// SIMATIC STEP 7 (V5.x) project cc1_15_7_14
// CPU: CPU 315-2 DP
// station: P_ADR_BUS
// station: Hardware
// station: SIMATIC 300 - BEC
// program: S7 Program(1)

FUNCTION FC 1 : VOID
AUTHOR : Arun
VERSION : 0.1
BEGIN
// (block stored without names or comments; labels and parameter names are numbered)
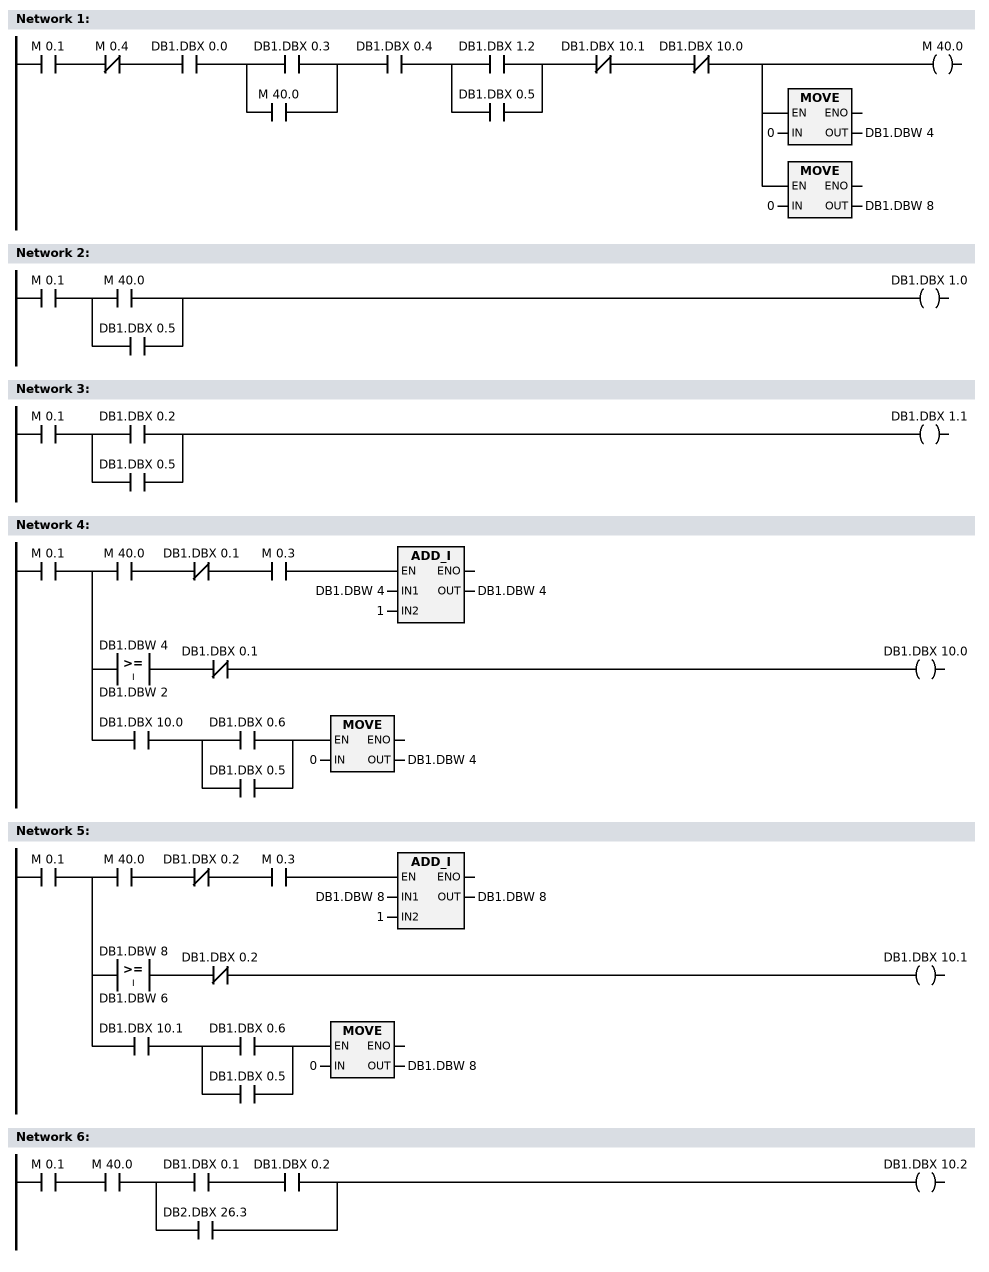
NETWORK
TITLE =
      A     M 0.1;
      AN    M 0.4;
      A     DB1.DBX 0.0;
      A(;
      O     DB1.DBX 0.3;
      O     M 40.0;
      );
      A     DB1.DBX 0.4;
      A(;
      O     DB1.DBX 1.2;
      O     DB1.DBX 0.5;
      );
      AN    DB1.DBX 10.1;
      AN    DB1.DBX 10.0;
      =     L 0.0;
      A     L 0.0;
      BLD   102;
      =     M 40.0;
      A     L 0.0;
      JNB   M001;
      L     0;
      T     DB1.DBW 4;
M001: NOP   0;
      A     L 0.0;
      JNB   M002;
      L     0;
      T     DB1.DBW 8;
M002: NOP   0;
NETWORK
TITLE =
      A     M 0.1;
      A(;
      O     M 40.0;
      O     DB1.DBX 0.5;
      );
      =     DB1.DBX 1.0;
NETWORK
TITLE =
      A     M 0.1;
      A(;
      O     DB1.DBX 0.2;
      O     DB1.DBX 0.5;
      );
      =     DB1.DBX 1.1;
NETWORK
TITLE =
      A     M 0.1;
      =     L 0.0;
      A     L 0.0;
      A     M 40.0;
      AN    DB1.DBX 0.1;
      A     M 0.3;
      JNB   M003;
      L     DB1.DBW 4;
      L     1;
      +I;
      T     DB1.DBW 4;
M003: NOP   0;
      A     L 0.0;
      A(;
      L     DB1.DBW 4;
      L     DB1.DBW 2;
      >=I;
      );
      AN    DB1.DBX 0.1;
      =     DB1.DBX 10.0;
      A     L 0.0;
      A     DB1.DBX 10.0;
      A(;
      O     DB1.DBX 0.6;
      O     DB1.DBX 0.5;
      );
      JNB   M004;
      L     0;
      T     DB1.DBW 4;
M004: NOP   0;
NETWORK
TITLE =
      A     M 0.1;
      =     L 0.0;
      A     L 0.0;
      A     M 40.0;
      AN    DB1.DBX 0.2;
      A     M 0.3;
      JNB   M005;
      L     DB1.DBW 8;
      L     1;
      +I;
      T     DB1.DBW 8;
M005: NOP   0;
      A     L 0.0;
      A(;
      L     DB1.DBW 8;
      L     DB1.DBW 6;
      >=I;
      );
      AN    DB1.DBX 0.2;
      =     DB1.DBX 10.1;
      A     L 0.0;
      A     DB1.DBX 10.1;
      A(;
      O     DB1.DBX 0.6;
      O     DB1.DBX 0.5;
      );
      JNB   M006;
      L     0;
      T     DB1.DBW 8;
M006: NOP   0;
NETWORK
TITLE =
      A     M 0.1;
      A     M 40.0;
      A(;
      A     DB1.DBX 0.1;
      A     DB1.DBX 0.2;
      O     DB2.DBX 26.3;
      );
      =     DB1.DBX 10.2;
END_FUNCTION

// FC 2: know-how protected block, not included

// FC 3: know-how protected block, not included

// FC 4: know-how protected block, not included

FUNCTION FC 5 : VOID
AUTHOR : Arun_Ram
VERSION : 0.1
BEGIN
// (block stored without names or comments; labels and parameter names are numbered)
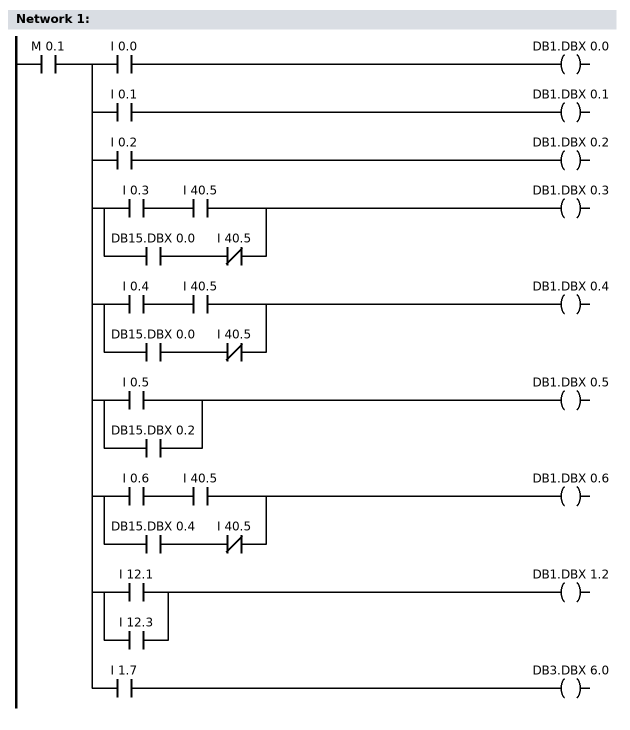
NETWORK
TITLE =
      A     M 0.1;
      =     L 0.0;
      A     L 0.0;
      A     I 0.0;
      =     DB1.DBX 0.0;
      A     L 0.0;
      A     I 0.1;
      =     DB1.DBX 0.1;
      A     L 0.0;
      A     I 0.2;
      =     DB1.DBX 0.2;
      A     L 0.0;
      A(;
      A     I 0.3;
      A     I 40.5;
      O;
      A     DB15.DBX 0.0;
      AN    I 40.5;
      );
      =     DB1.DBX 0.3;
      A     L 0.0;
      A(;
      A     I 0.4;
      A     I 40.5;
      O;
      A     DB15.DBX 0.0;
      AN    I 40.5;
      );
      =     DB1.DBX 0.4;
      A     L 0.0;
      A(;
      O     I 0.5;
      O     DB15.DBX 0.2;
      );
      =     DB1.DBX 0.5;
      A     L 0.0;
      A(;
      A     I 0.6;
      A     I 40.5;
      O;
      A     DB15.DBX 0.4;
      AN    I 40.5;
      );
      =     DB1.DBX 0.6;
      A     L 0.0;
      A(;
      O     I 12.1;
      O     I 12.3;
      );
      =     DB1.DBX 1.2;
      A     L 0.0;
      A     I 1.7;
      =     DB3.DBX 6.0;
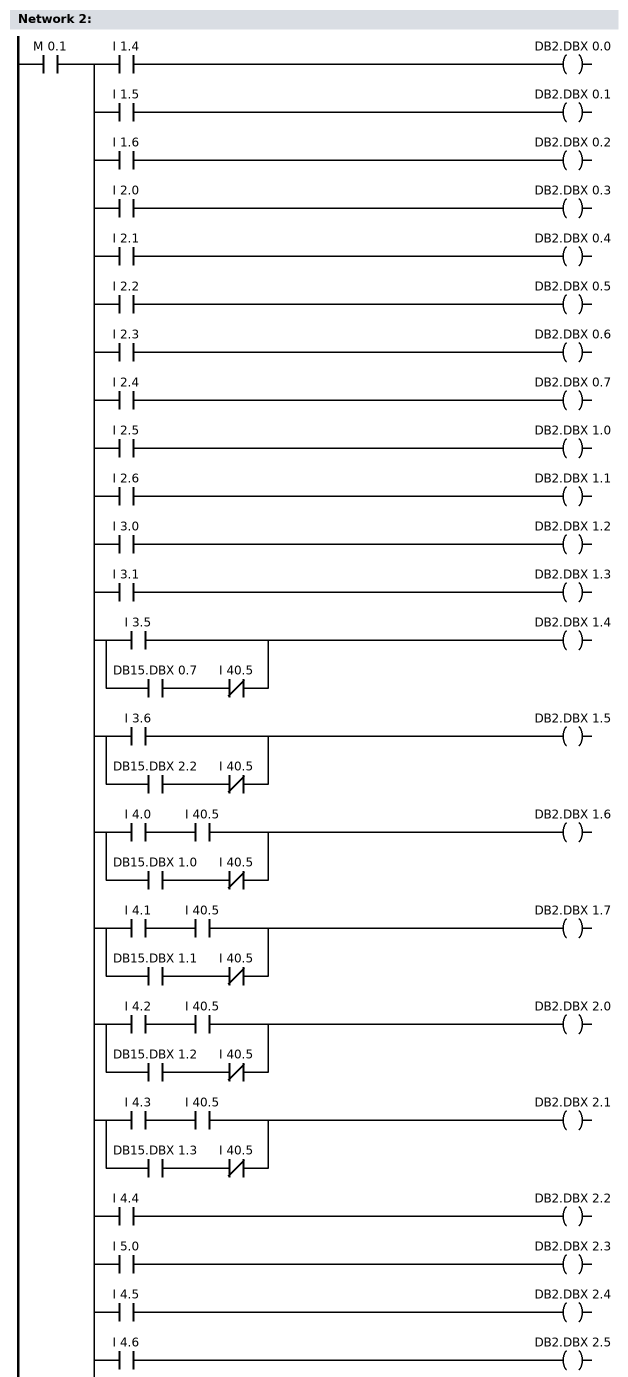
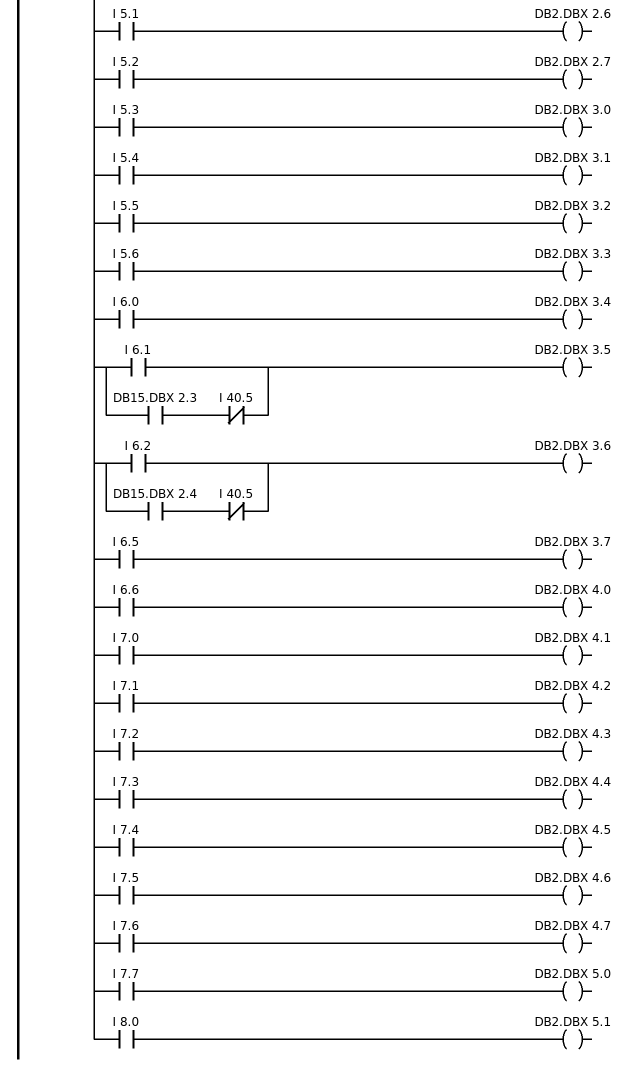
NETWORK
TITLE =
      A     M 0.1;
      =     L 0.0;
      A     L 0.0;
      A     I 1.4;
      =     DB2.DBX 0.0;
      A     L 0.0;
      A     I 1.5;
      =     DB2.DBX 0.1;
      A     L 0.0;
      A     I 1.6;
      =     DB2.DBX 0.2;
      A     L 0.0;
      A     I 2.0;
      =     DB2.DBX 0.3;
      A     L 0.0;
      A     I 2.1;
      =     DB2.DBX 0.4;
      A     L 0.0;
      A     I 2.2;
      =     DB2.DBX 0.5;
      A     L 0.0;
      A     I 2.3;
      =     DB2.DBX 0.6;
      A     L 0.0;
      A     I 2.4;
      =     DB2.DBX 0.7;
      A     L 0.0;
      A     I 2.5;
      =     DB2.DBX 1.0;
      A     L 0.0;
      A     I 2.6;
      =     DB2.DBX 1.1;
      A     L 0.0;
      A     I 3.0;
      =     DB2.DBX 1.2;
      A     L 0.0;
      A     I 3.1;
      =     DB2.DBX 1.3;
      A     L 0.0;
      A(;
      O     I 3.5;
      O;
      A     DB15.DBX 0.7;
      AN    I 40.5;
      );
      =     DB2.DBX 1.4;
      A     L 0.0;
      A(;
      O     I 3.6;
      O;
      A     DB15.DBX 2.2;
      AN    I 40.5;
      );
      =     DB2.DBX 1.5;
      A     L 0.0;
      A(;
      A     I 4.0;
      A     I 40.5;
      O;
      A     DB15.DBX 1.0;
      AN    I 40.5;
      );
      =     DB2.DBX 1.6;
      A     L 0.0;
      A(;
      A     I 4.1;
      A     I 40.5;
      O;
      A     DB15.DBX 1.1;
      AN    I 40.5;
      );
      =     DB2.DBX 1.7;
      A     L 0.0;
      A(;
      A     I 4.2;
      A     I 40.5;
      O;
      A     DB15.DBX 1.2;
      AN    I 40.5;
      );
      =     DB2.DBX 2.0;
      A     L 0.0;
      A(;
      A     I 4.3;
      A     I 40.5;
      O;
      A     DB15.DBX 1.3;
      AN    I 40.5;
      );
      =     DB2.DBX 2.1;
      A     L 0.0;
      A     I 4.4;
      =     DB2.DBX 2.2;
      A     L 0.0;
      A     I 5.0;
      =     DB2.DBX 2.3;
      A     L 0.0;
      A     I 4.5;
      =     DB2.DBX 2.4;
      A     L 0.0;
      A     I 4.6;
      =     DB2.DBX 2.5;
      A     L 0.0;
      A     I 5.1;
      =     DB2.DBX 2.6;
      A     L 0.0;
      A     I 5.2;
      =     DB2.DBX 2.7;
      A     L 0.0;
      A     I 5.3;
      =     DB2.DBX 3.0;
      A     L 0.0;
      A     I 5.4;
      =     DB2.DBX 3.1;
      A     L 0.0;
      A     I 5.5;
      =     DB2.DBX 3.2;
      A     L 0.0;
      A     I 5.6;
      =     DB2.DBX 3.3;
      A     L 0.0;
      A     I 6.0;
      =     DB2.DBX 3.4;
      A     L 0.0;
      A(;
      O     I 6.1;
      O;
      A     DB15.DBX 2.3;
      AN    I 40.5;
      );
      =     DB2.DBX 3.5;
      A     L 0.0;
      A(;
      O     I 6.2;
      O;
      A     DB15.DBX 2.4;
      AN    I 40.5;
      );
      =     DB2.DBX 3.6;
      A     L 0.0;
      A     I 6.5;
      =     DB2.DBX 3.7;
      A     L 0.0;
      A     I 6.6;
      =     DB2.DBX 4.0;
      A     L 0.0;
      A     I 7.0;
      =     DB2.DBX 4.1;
      A     L 0.0;
      A     I 7.1;
      =     DB2.DBX 4.2;
      A     L 0.0;
      A     I 7.2;
      =     DB2.DBX 4.3;
      A     L 0.0;
      A     I 7.3;
      =     DB2.DBX 4.4;
      A     L 0.0;
      A     I 7.4;
      =     DB2.DBX 4.5;
      A     L 0.0;
      A     I 7.5;
      =     DB2.DBX 4.6;
      A     L 0.0;
      A     I 7.6;
      =     DB2.DBX 4.7;
      A     L 0.0;
      A     I 7.7;
      =     DB2.DBX 5.0;
      A     L 0.0;
      A     I 8.0;
      =     DB2.DBX 5.1;
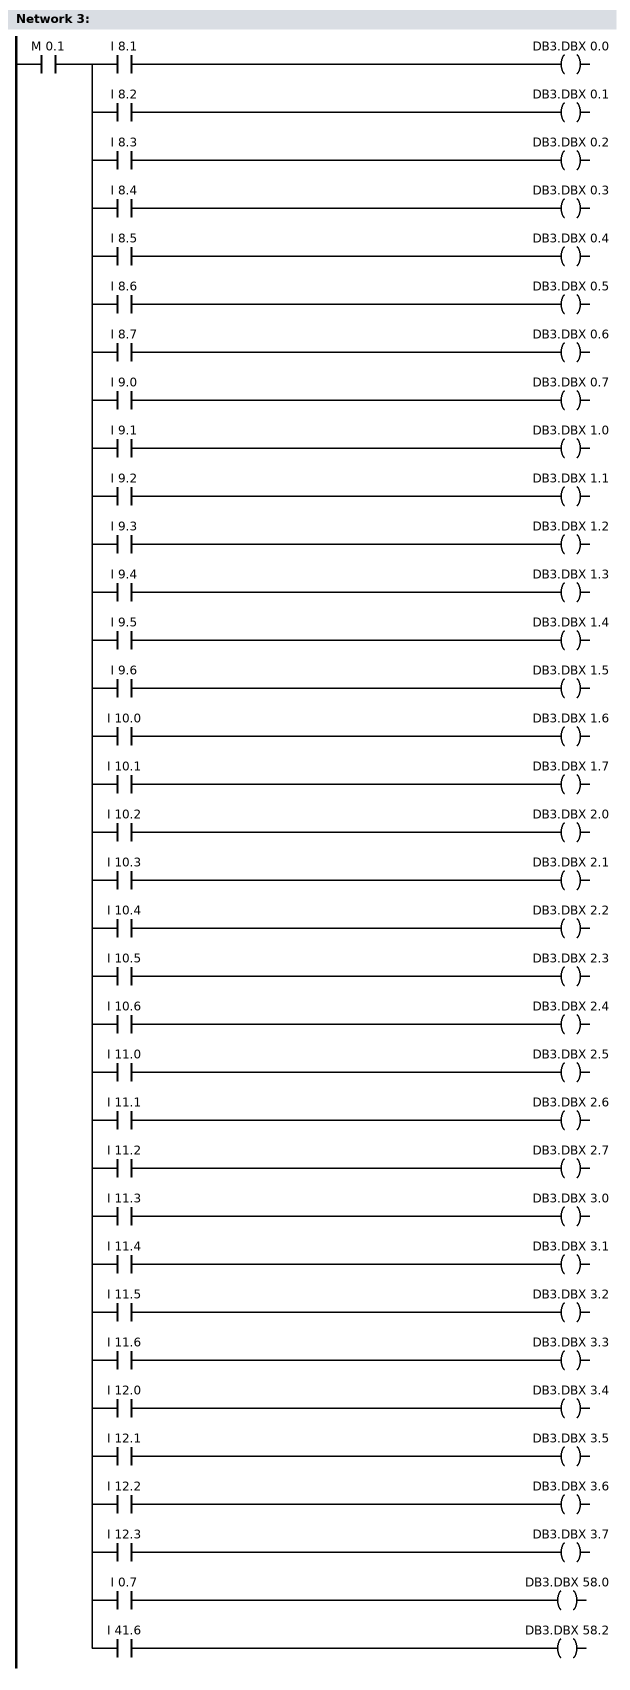
NETWORK
TITLE =
      A     M 0.1;
      =     L 0.0;
      A     L 0.0;
      A     I 8.1;
      =     DB3.DBX 0.0;
      A     L 0.0;
      A     I 8.2;
      =     DB3.DBX 0.1;
      A     L 0.0;
      A     I 8.3;
      =     DB3.DBX 0.2;
      A     L 0.0;
      A     I 8.4;
      =     DB3.DBX 0.3;
      A     L 0.0;
      A     I 8.5;
      =     DB3.DBX 0.4;
      A     L 0.0;
      A     I 8.6;
      =     DB3.DBX 0.5;
      A     L 0.0;
      A     I 8.7;
      =     DB3.DBX 0.6;
      A     L 0.0;
      A     I 9.0;
      =     DB3.DBX 0.7;
      A     L 0.0;
      A     I 9.1;
      =     DB3.DBX 1.0;
      A     L 0.0;
      A     I 9.2;
      =     DB3.DBX 1.1;
      A     L 0.0;
      A     I 9.3;
      =     DB3.DBX 1.2;
      A     L 0.0;
      A     I 9.4;
      =     DB3.DBX 1.3;
      A     L 0.0;
      A     I 9.5;
      =     DB3.DBX 1.4;
      A     L 0.0;
      A     I 9.6;
      =     DB3.DBX 1.5;
      A     L 0.0;
      A     I 10.0;
      =     DB3.DBX 1.6;
      A     L 0.0;
      A     I 10.1;
      =     DB3.DBX 1.7;
      A     L 0.0;
      A     I 10.2;
      =     DB3.DBX 2.0;
      A     L 0.0;
      A     I 10.3;
      =     DB3.DBX 2.1;
      A     L 0.0;
      A     I 10.4;
      =     DB3.DBX 2.2;
      A     L 0.0;
      A     I 10.5;
      =     DB3.DBX 2.3;
      A     L 0.0;
      A     I 10.6;
      =     DB3.DBX 2.4;
      A     L 0.0;
      A     I 11.0;
      =     DB3.DBX 2.5;
      A     L 0.0;
      A     I 11.1;
      =     DB3.DBX 2.6;
      A     L 0.0;
      A     I 11.2;
      =     DB3.DBX 2.7;
      A     L 0.0;
      A     I 11.3;
      =     DB3.DBX 3.0;
      A     L 0.0;
      A     I 11.4;
      =     DB3.DBX 3.1;
      A     L 0.0;
      A     I 11.5;
      =     DB3.DBX 3.2;
      A     L 0.0;
      A     I 11.6;
      =     DB3.DBX 3.3;
      A     L 0.0;
      A     I 12.0;
      =     DB3.DBX 3.4;
      A     L 0.0;
      A     I 12.1;
      =     DB3.DBX 3.5;
      A     L 0.0;
      A     I 12.2;
      =     DB3.DBX 3.6;
      A     L 0.0;
      A     I 12.3;
      =     DB3.DBX 3.7;
      A     L 0.0;
      A     I 0.7;
      =     DB3.DBX 58.0;
      A     L 0.0;
      A     I 41.6;
      =     DB3.DBX 58.2;
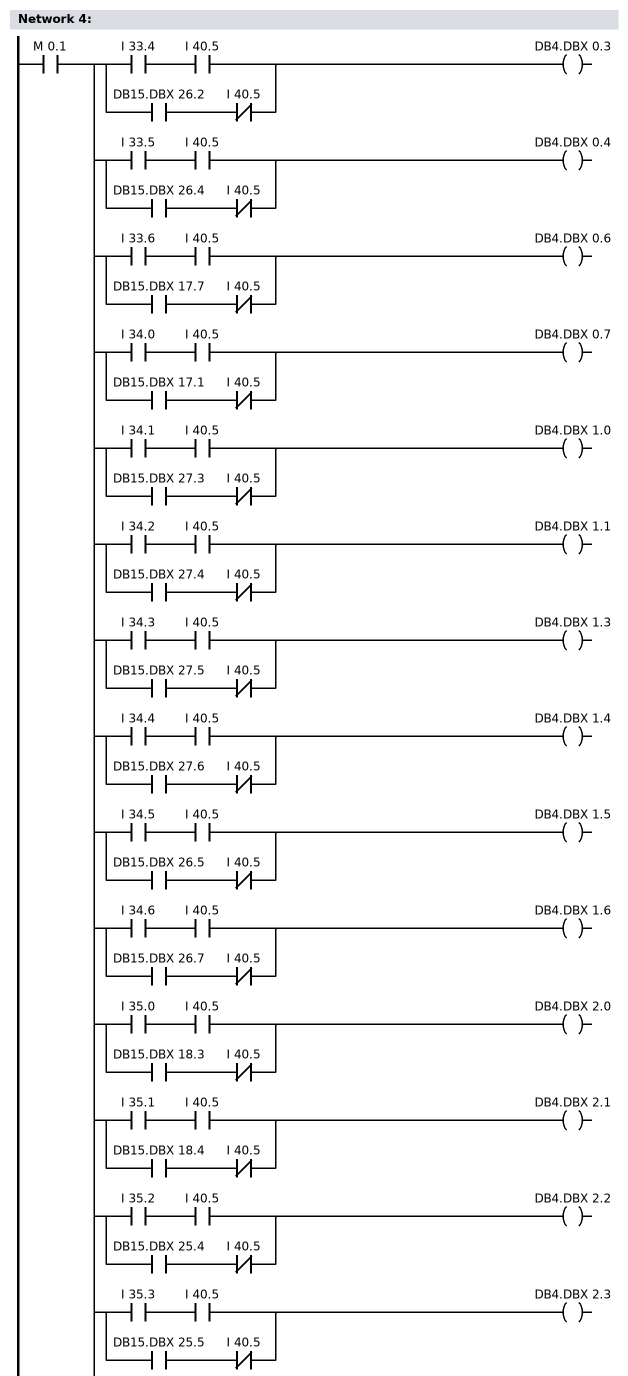
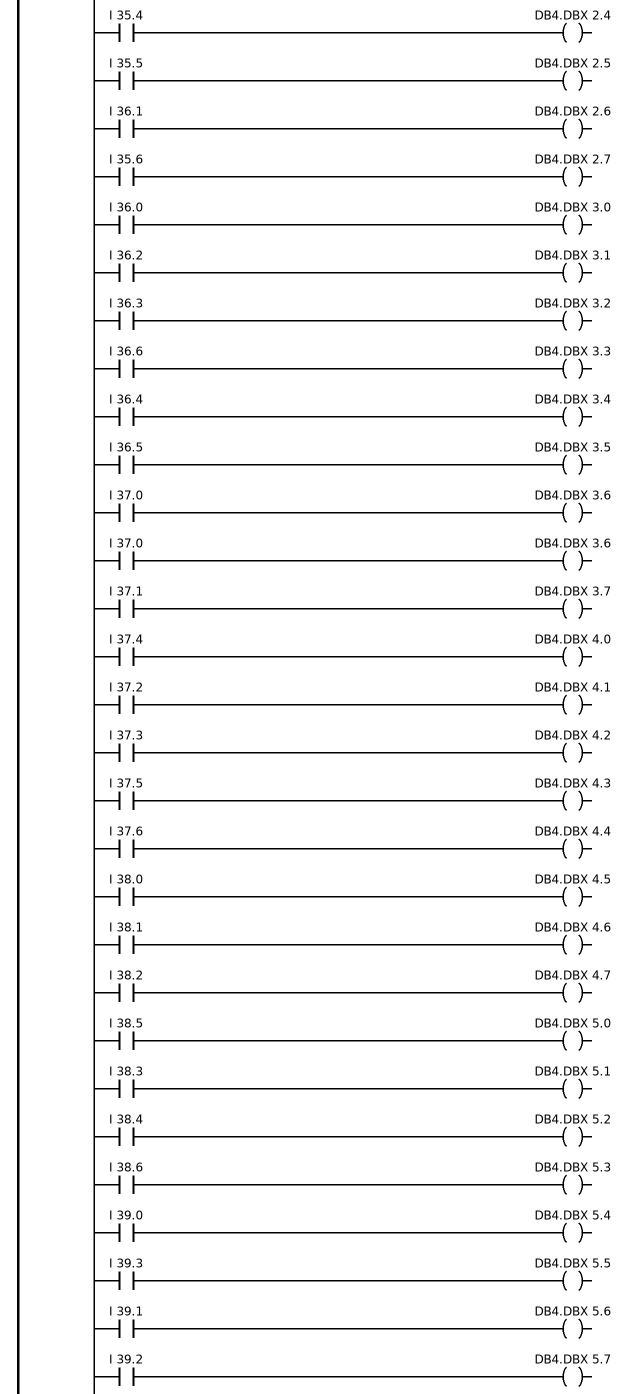
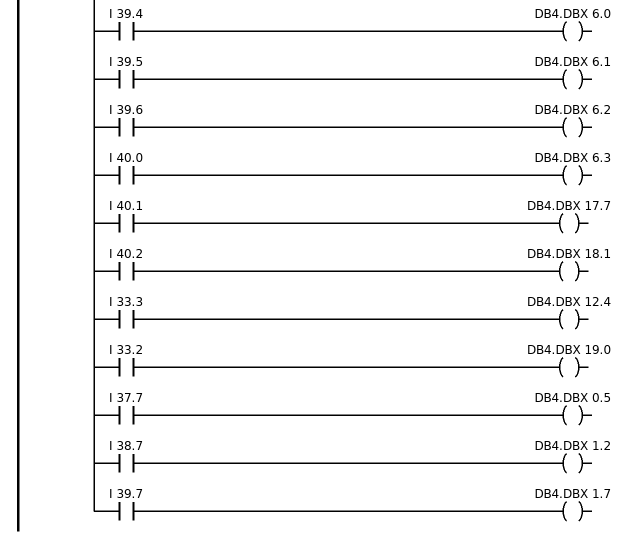
NETWORK
TITLE =
      A     M 0.1;
      =     L 0.0;
      A     L 0.0;
      A(;
      A     I 33.4;
      A     I 40.5;
      O;
      A     DB15.DBX 26.2;
      AN    I 40.5;
      );
      =     DB4.DBX 0.3;
      A     L 0.0;
      A(;
      A     I 33.5;
      A     I 40.5;
      O;
      A     DB15.DBX 26.4;
      AN    I 40.5;
      );
      =     DB4.DBX 0.4;
      A     L 0.0;
      A(;
      A     I 33.6;
      A     I 40.5;
      O;
      A     DB15.DBX 17.7;
      AN    I 40.5;
      );
      =     DB4.DBX 0.6;
      A     L 0.0;
      A(;
      A     I 34.0;
      A     I 40.5;
      O;
      A     DB15.DBX 17.1;
      AN    I 40.5;
      );
      =     DB4.DBX 0.7;
      A     L 0.0;
      A(;
      A     I 34.1;
      A     I 40.5;
      O;
      A     DB15.DBX 27.3;
      AN    I 40.5;
      );
      =     DB4.DBX 1.0;
      A     L 0.0;
      A(;
      A     I 34.2;
      A     I 40.5;
      O;
      A     DB15.DBX 27.4;
      AN    I 40.5;
      );
      =     DB4.DBX 1.1;
      A     L 0.0;
      A(;
      A     I 34.3;
      A     I 40.5;
      O;
      A     DB15.DBX 27.5;
      AN    I 40.5;
      );
      =     DB4.DBX 1.3;
      A     L 0.0;
      A(;
      A     I 34.4;
      A     I 40.5;
      O;
      A     DB15.DBX 27.6;
      AN    I 40.5;
      );
      =     DB4.DBX 1.4;
      A     L 0.0;
      A(;
      A     I 34.5;
      A     I 40.5;
      O;
      A     DB15.DBX 26.5;
      AN    I 40.5;
      );
      =     DB4.DBX 1.5;
      A     L 0.0;
      A(;
      A     I 34.6;
      A     I 40.5;
      O;
      A     DB15.DBX 26.7;
      AN    I 40.5;
      );
      =     DB4.DBX 1.6;
      A     L 0.0;
      A(;
      A     I 35.0;
      A     I 40.5;
      O;
      A     DB15.DBX 18.3;
      AN    I 40.5;
      );
      =     DB4.DBX 2.0;
      A     L 0.0;
      A(;
      A     I 35.1;
      A     I 40.5;
      O;
      A     DB15.DBX 18.4;
      AN    I 40.5;
      );
      =     DB4.DBX 2.1;
      A     L 0.0;
      A(;
      A     I 35.2;
      A     I 40.5;
      O;
      A     DB15.DBX 25.4;
      AN    I 40.5;
      );
      =     DB4.DBX 2.2;
      A     L 0.0;
      A(;
      A     I 35.3;
      A     I 40.5;
      O;
      A     DB15.DBX 25.5;
      AN    I 40.5;
      );
      =     DB4.DBX 2.3;
      A     L 0.0;
      A     I 35.4;
      =     DB4.DBX 2.4;
      A     L 0.0;
      A     I 35.5;
      =     DB4.DBX 2.5;
      A     L 0.0;
      A     I 36.1;
      =     DB4.DBX 2.6;
      A     L 0.0;
      A     I 35.6;
      =     DB4.DBX 2.7;
      A     L 0.0;
      A     I 36.0;
      =     DB4.DBX 3.0;
      A     L 0.0;
      A     I 36.2;
      =     DB4.DBX 3.1;
      A     L 0.0;
      A     I 36.3;
      =     DB4.DBX 3.2;
      A     L 0.0;
      A     I 36.6;
      =     DB4.DBX 3.3;
      A     L 0.0;
      A     I 36.4;
      =     DB4.DBX 3.4;
      A     L 0.0;
      A     I 36.5;
      =     DB4.DBX 3.5;
      A     L 0.0;
      A     I 37.0;
      =     DB4.DBX 3.6;
      A     L 0.0;
      A     I 37.0;
      =     DB4.DBX 3.6;
      A     L 0.0;
      A     I 37.1;
      =     DB4.DBX 3.7;
      A     L 0.0;
      A     I 37.4;
      =     DB4.DBX 4.0;
      A     L 0.0;
      A     I 37.2;
      =     DB4.DBX 4.1;
      A     L 0.0;
      A     I 37.3;
      =     DB4.DBX 4.2;
      A     L 0.0;
      A     I 37.5;
      =     DB4.DBX 4.3;
      A     L 0.0;
      A     I 37.6;
      =     DB4.DBX 4.4;
      A     L 0.0;
      A     I 38.0;
      =     DB4.DBX 4.5;
      A     L 0.0;
      A     I 38.1;
      =     DB4.DBX 4.6;
      A     L 0.0;
      A     I 38.2;
      =     DB4.DBX 4.7;
      A     L 0.0;
      A     I 38.5;
      =     DB4.DBX 5.0;
      A     L 0.0;
      A     I 38.3;
      =     DB4.DBX 5.1;
      A     L 0.0;
      A     I 38.4;
      =     DB4.DBX 5.2;
      A     L 0.0;
      A     I 38.6;
      =     DB4.DBX 5.3;
      A     L 0.0;
      A     I 39.0;
      =     DB4.DBX 5.4;
      A     L 0.0;
      A     I 39.3;
      =     DB4.DBX 5.5;
      A     L 0.0;
      A     I 39.1;
      =     DB4.DBX 5.6;
      A     L 0.0;
      A     I 39.2;
      =     DB4.DBX 5.7;
      A     L 0.0;
      A     I 39.4;
      =     DB4.DBX 6.0;
      A     L 0.0;
      A     I 39.5;
      =     DB4.DBX 6.1;
      A     L 0.0;
      A     I 39.6;
      =     DB4.DBX 6.2;
      A     L 0.0;
      A     I 40.0;
      =     DB4.DBX 6.3;
      A     L 0.0;
      A     I 40.1;
      =     DB4.DBX 17.7;
      A     L 0.0;
      A     I 40.2;
      =     DB4.DBX 18.1;
      A     L 0.0;
      A     I 33.3;
      =     DB4.DBX 12.4;
      A     L 0.0;
      A     I 33.2;
      =     DB4.DBX 19.0;
      A     L 0.0;
      A     I 37.7;
      =     DB4.DBX 0.5;
      A     L 0.0;
      A     I 38.7;
      =     DB4.DBX 1.2;
      A     L 0.0;
      A     I 39.7;
      =     DB4.DBX 1.7;
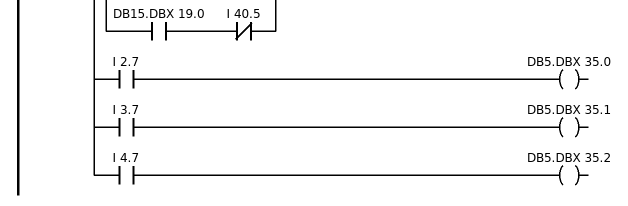
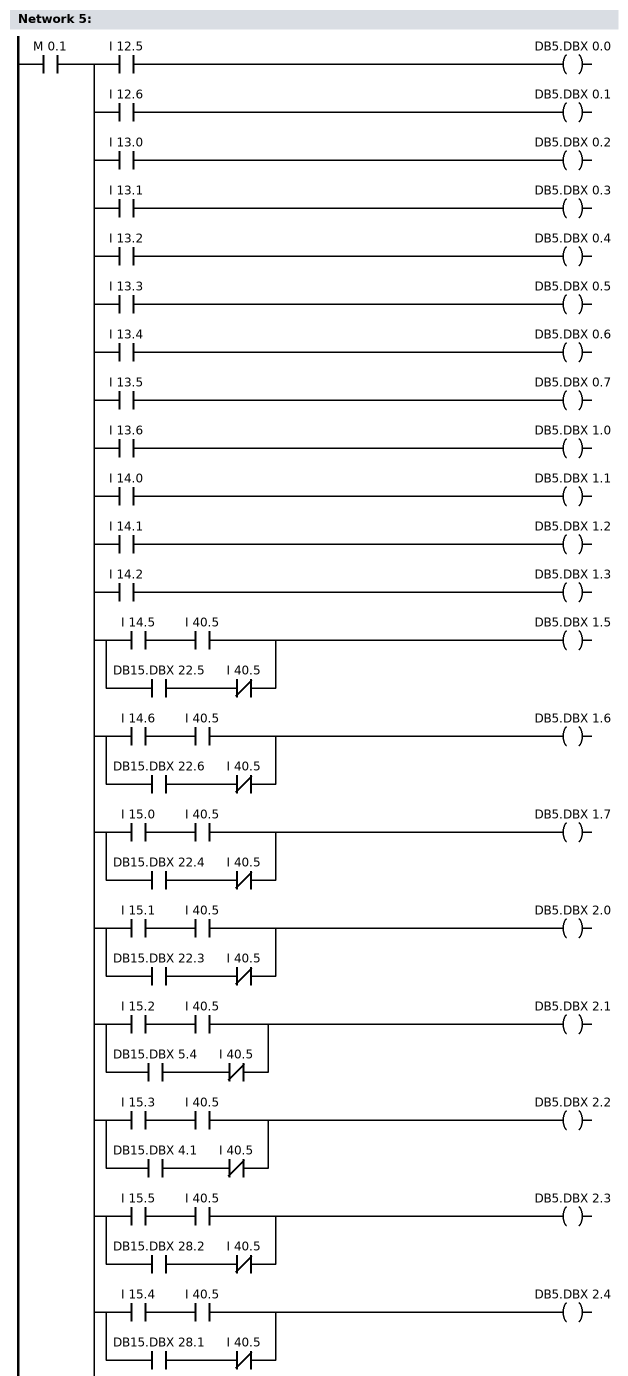
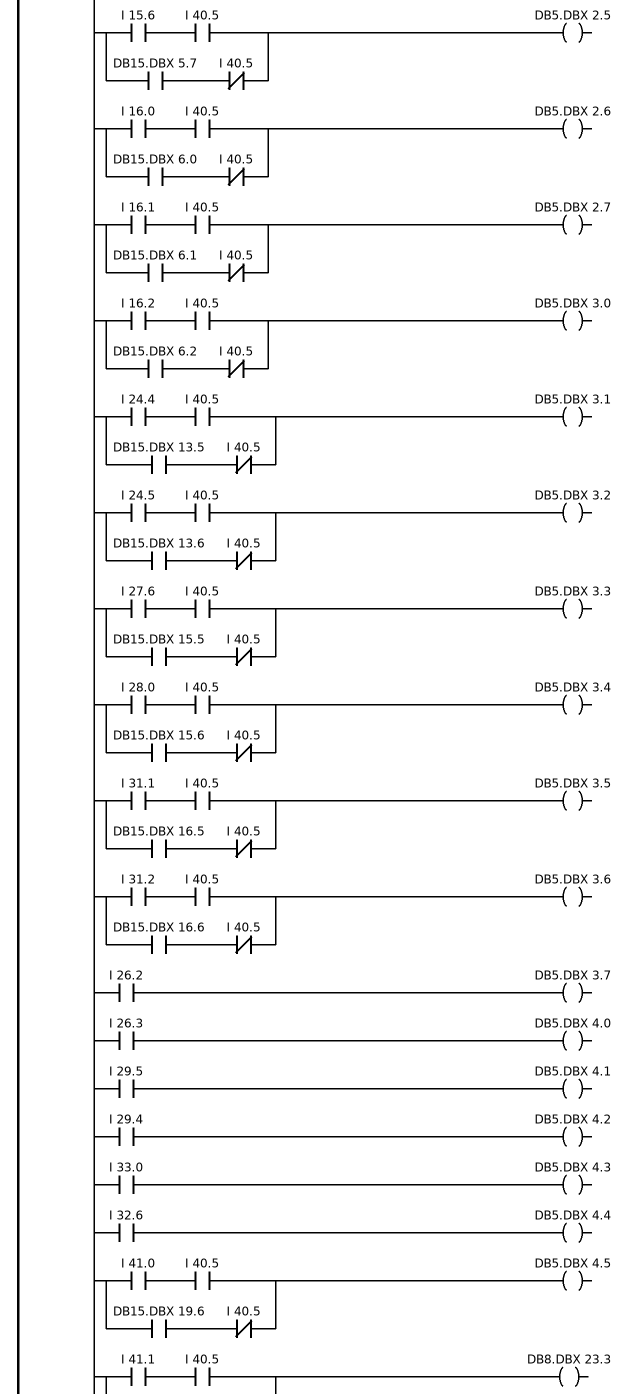
NETWORK
TITLE =
      A     M 0.1;
      =     L 0.0;
      A     L 0.0;
      A     I 12.5;
      =     DB5.DBX 0.0;
      A     L 0.0;
      A     I 12.6;
      =     DB5.DBX 0.1;
      A     L 0.0;
      A     I 13.0;
      =     DB5.DBX 0.2;
      A     L 0.0;
      A     I 13.1;
      =     DB5.DBX 0.3;
      A     L 0.0;
      A     I 13.2;
      =     DB5.DBX 0.4;
      A     L 0.0;
      A     I 13.3;
      =     DB5.DBX 0.5;
      A     L 0.0;
      A     I 13.4;
      =     DB5.DBX 0.6;
      A     L 0.0;
      A     I 13.5;
      =     DB5.DBX 0.7;
      A     L 0.0;
      A     I 13.6;
      =     DB5.DBX 1.0;
      A     L 0.0;
      A     I 14.0;
      =     DB5.DBX 1.1;
      A     L 0.0;
      A     I 14.1;
      =     DB5.DBX 1.2;
      A     L 0.0;
      A     I 14.2;
      =     DB5.DBX 1.3;
      A     L 0.0;
      A(;
      A     I 14.5;
      A     I 40.5;
      O;
      A     DB15.DBX 22.5;
      AN    I 40.5;
      );
      =     DB5.DBX 1.5;
      A     L 0.0;
      A(;
      A     I 14.6;
      A     I 40.5;
      O;
      A     DB15.DBX 22.6;
      AN    I 40.5;
      );
      =     DB5.DBX 1.6;
      A     L 0.0;
      A(;
      A     I 15.0;
      A     I 40.5;
      O;
      A     DB15.DBX 22.4;
      AN    I 40.5;
      );
      =     DB5.DBX 1.7;
      A     L 0.0;
      A(;
      A     I 15.1;
      A     I 40.5;
      O;
      A     DB15.DBX 22.3;
      AN    I 40.5;
      );
      =     DB5.DBX 2.0;
      A     L 0.0;
      A(;
      A     I 15.2;
      A     I 40.5;
      O;
      A     DB15.DBX 5.4;
      AN    I 40.5;
      );
      =     DB5.DBX 2.1;
      A     L 0.0;
      A(;
      A     I 15.3;
      A     I 40.5;
      O;
      A     DB15.DBX 4.1;
      AN    I 40.5;
      );
      =     DB5.DBX 2.2;
      A     L 0.0;
      A(;
      A     I 15.5;
      A     I 40.5;
      O;
      A     DB15.DBX 28.2;
      AN    I 40.5;
      );
      =     DB5.DBX 2.3;
      A     L 0.0;
      A(;
      A     I 15.4;
      A     I 40.5;
      O;
      A     DB15.DBX 28.1;
      AN    I 40.5;
      );
      =     DB5.DBX 2.4;
      A     L 0.0;
      A(;
      A     I 15.6;
      A     I 40.5;
      O;
      A     DB15.DBX 5.7;
      AN    I 40.5;
      );
      =     DB5.DBX 2.5;
      A     L 0.0;
      A(;
      A     I 16.0;
      A     I 40.5;
      O;
      A     DB15.DBX 6.0;
      AN    I 40.5;
      );
      =     DB5.DBX 2.6;
      A     L 0.0;
      A(;
      A     I 16.1;
      A     I 40.5;
      O;
      A     DB15.DBX 6.1;
      AN    I 40.5;
      );
      =     DB5.DBX 2.7;
      A     L 0.0;
      A(;
      A     I 16.2;
      A     I 40.5;
      O;
      A     DB15.DBX 6.2;
      AN    I 40.5;
      );
      =     DB5.DBX 3.0;
      A     L 0.0;
      A(;
      A     I 24.4;
      A     I 40.5;
      O;
      A     DB15.DBX 13.5;
      AN    I 40.5;
      );
      =     DB5.DBX 3.1;
      A     L 0.0;
      A(;
      A     I 24.5;
      A     I 40.5;
      O;
      A     DB15.DBX 13.6;
      AN    I 40.5;
      );
      =     DB5.DBX 3.2;
      A     L 0.0;
      A(;
      A     I 27.6;
      A     I 40.5;
      O;
      A     DB15.DBX 15.5;
      AN    I 40.5;
      );
      =     DB5.DBX 3.3;
      A     L 0.0;
      A(;
      A     I 28.0;
      A     I 40.5;
      O;
      A     DB15.DBX 15.6;
      AN    I 40.5;
      );
      =     DB5.DBX 3.4;
      A     L 0.0;
      A(;
      A     I 31.1;
      A     I 40.5;
      O;
      A     DB15.DBX 16.5;
      AN    I 40.5;
      );
      =     DB5.DBX 3.5;
      A     L 0.0;
      A(;
      A     I 31.2;
      A     I 40.5;
      O;
      A     DB15.DBX 16.6;
      AN    I 40.5;
      );
      =     DB5.DBX 3.6;
      A     L 0.0;
      A     I 26.2;
      =     DB5.DBX 3.7;
      A     L 0.0;
      A     I 26.3;
      =     DB5.DBX 4.0;
      A     L 0.0;
      A     I 29.5;
      =     DB5.DBX 4.1;
      A     L 0.0;
      A     I 29.4;
      =     DB5.DBX 4.2;
      A     L 0.0;
      A     I 33.0;
      =     DB5.DBX 4.3;
      A     L 0.0;
      A     I 32.6;
      =     DB5.DBX 4.4;
      A     L 0.0;
      A(;
      A     I 41.0;
      A     I 40.5;
      O;
      A     DB15.DBX 19.6;
      AN    I 40.5;
      );
      =     DB5.DBX 4.5;
      A     L 0.0;
      A(;
      A     I 41.1;
      A     I 40.5;
      O;
      A     DB15.DBX 19.0;
      AN    I 40.5;
      );
      =     DB8.DBX 23.3;
      A     L 0.0;
      A     I 2.7;
      =     DB5.DBX 35.0;
      A     L 0.0;
      A     I 3.7;
      =     DB5.DBX 35.1;
      A     L 0.0;
      A     I 4.7;
      =     DB5.DBX 35.2;
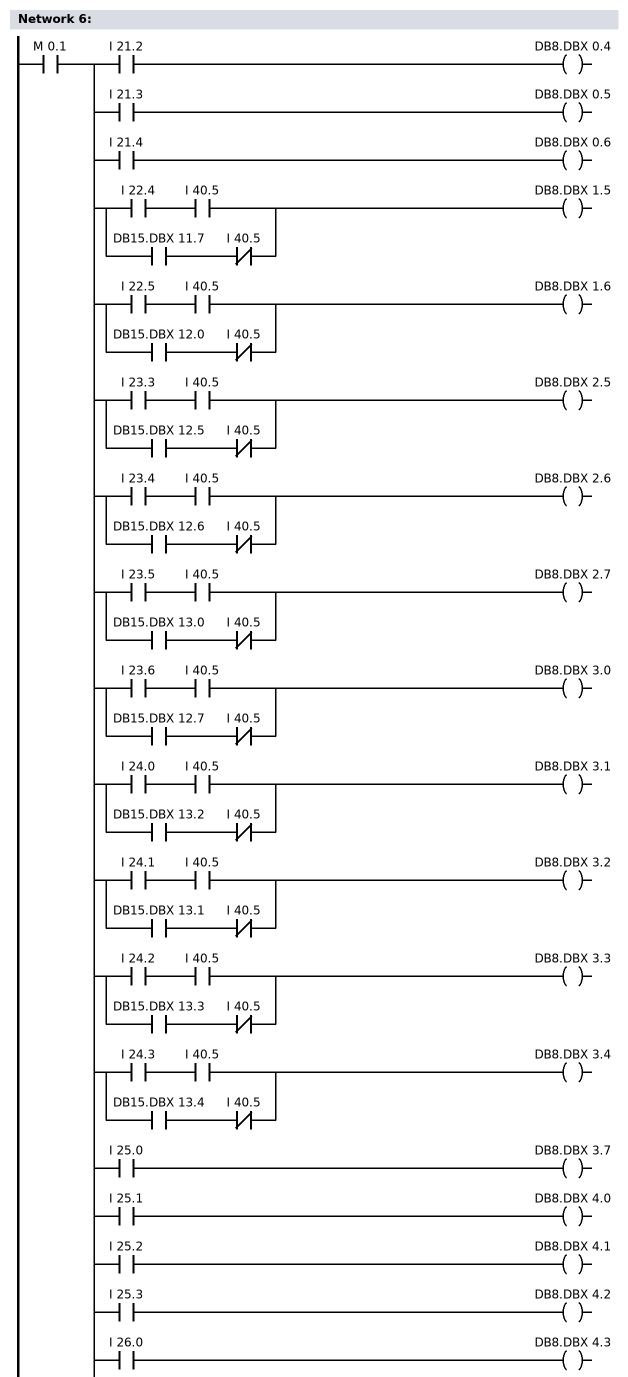
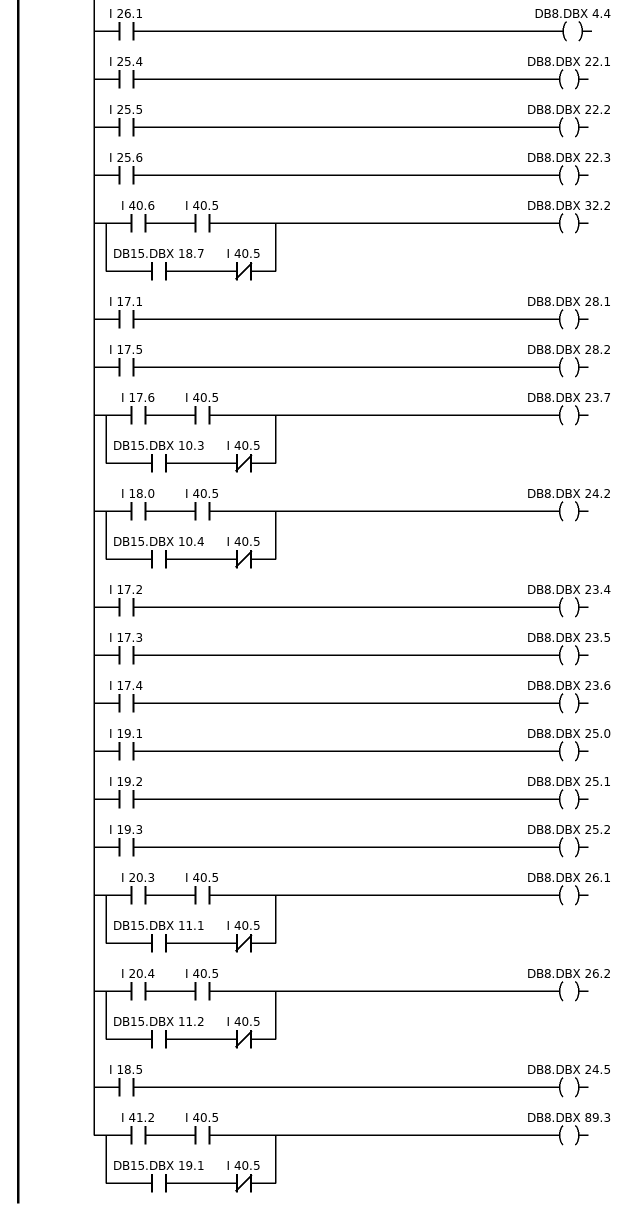
NETWORK
TITLE =
      A     M 0.1;
      =     L 0.0;
      A     L 0.0;
      A     I 21.2;
      =     DB8.DBX 0.4;
      A     L 0.0;
      A     I 21.3;
      =     DB8.DBX 0.5;
      A     L 0.0;
      A     I 21.4;
      =     DB8.DBX 0.6;
      A     L 0.0;
      A(;
      A     I 22.4;
      A     I 40.5;
      O;
      A     DB15.DBX 11.7;
      AN    I 40.5;
      );
      =     DB8.DBX 1.5;
      A     L 0.0;
      A(;
      A     I 22.5;
      A     I 40.5;
      O;
      A     DB15.DBX 12.0;
      AN    I 40.5;
      );
      =     DB8.DBX 1.6;
      A     L 0.0;
      A(;
      A     I 23.3;
      A     I 40.5;
      O;
      A     DB15.DBX 12.5;
      AN    I 40.5;
      );
      =     DB8.DBX 2.5;
      A     L 0.0;
      A(;
      A     I 23.4;
      A     I 40.5;
      O;
      A     DB15.DBX 12.6;
      AN    I 40.5;
      );
      =     DB8.DBX 2.6;
      A     L 0.0;
      A(;
      A     I 23.5;
      A     I 40.5;
      O;
      A     DB15.DBX 13.0;
      AN    I 40.5;
      );
      =     DB8.DBX 2.7;
      A     L 0.0;
      A(;
      A     I 23.6;
      A     I 40.5;
      O;
      A     DB15.DBX 12.7;
      AN    I 40.5;
      );
      =     DB8.DBX 3.0;
      A     L 0.0;
      A(;
      A     I 24.0;
      A     I 40.5;
      O;
      A     DB15.DBX 13.2;
      AN    I 40.5;
      );
      =     DB8.DBX 3.1;
      A     L 0.0;
      A(;
      A     I 24.1;
      A     I 40.5;
      O;
      A     DB15.DBX 13.1;
      AN    I 40.5;
      );
      =     DB8.DBX 3.2;
      A     L 0.0;
      A(;
      A     I 24.2;
      A     I 40.5;
      O;
      A     DB15.DBX 13.3;
      AN    I 40.5;
      );
      =     DB8.DBX 3.3;
      A     L 0.0;
      A(;
      A     I 24.3;
      A     I 40.5;
      O;
      A     DB15.DBX 13.4;
      AN    I 40.5;
      );
      =     DB8.DBX 3.4;
      A     L 0.0;
      A     I 25.0;
      =     DB8.DBX 3.7;
      A     L 0.0;
      A     I 25.1;
      =     DB8.DBX 4.0;
      A     L 0.0;
      A     I 25.2;
      =     DB8.DBX 4.1;
      A     L 0.0;
      A     I 25.3;
      =     DB8.DBX 4.2;
      A     L 0.0;
      A     I 26.0;
      =     DB8.DBX 4.3;
      A     L 0.0;
      A     I 26.1;
      =     DB8.DBX 4.4;
      A     L 0.0;
      A     I 25.4;
      =     DB8.DBX 22.1;
      A     L 0.0;
      A     I 25.5;
      =     DB8.DBX 22.2;
      A     L 0.0;
      A     I 25.6;
      =     DB8.DBX 22.3;
      A     L 0.0;
      A(;
      A     I 40.6;
      A     I 40.5;
      O;
      A     DB15.DBX 18.7;
      AN    I 40.5;
      );
      =     DB8.DBX 32.2;
      A     L 0.0;
      A     I 17.1;
      =     DB8.DBX 28.1;
      A     L 0.0;
      A     I 17.5;
      =     DB8.DBX 28.2;
      A     L 0.0;
      A(;
      A     I 17.6;
      A     I 40.5;
      O;
      A     DB15.DBX 10.3;
      AN    I 40.5;
      );
      =     DB8.DBX 23.7;
      A     L 0.0;
      A(;
      A     I 18.0;
      A     I 40.5;
      O;
      A     DB15.DBX 10.4;
      AN    I 40.5;
      );
      =     DB8.DBX 24.2;
      A     L 0.0;
      A     I 17.2;
      =     DB8.DBX 23.4;
      A     L 0.0;
      A     I 17.3;
      =     DB8.DBX 23.5;
      A     L 0.0;
      A     I 17.4;
      =     DB8.DBX 23.6;
      A     L 0.0;
      A     I 19.1;
      =     DB8.DBX 25.0;
      A     L 0.0;
      A     I 19.2;
      =     DB8.DBX 25.1;
      A     L 0.0;
      A     I 19.3;
      =     DB8.DBX 25.2;
      A     L 0.0;
      A(;
      A     I 20.3;
      A     I 40.5;
      O;
      A     DB15.DBX 11.1;
      AN    I 40.5;
      );
      =     DB8.DBX 26.1;
      A     L 0.0;
      A(;
      A     I 20.4;
      A     I 40.5;
      O;
      A     DB15.DBX 11.2;
      AN    I 40.5;
      );
      =     DB8.DBX 26.2;
      A     L 0.0;
      A     I 18.5;
      =     DB8.DBX 24.5;
      A     L 0.0;
      A(;
      A     I 41.2;
      A     I 40.5;
      O;
      A     DB15.DBX 19.1;
      AN    I 40.5;
      );
      =     DB8.DBX 89.3;
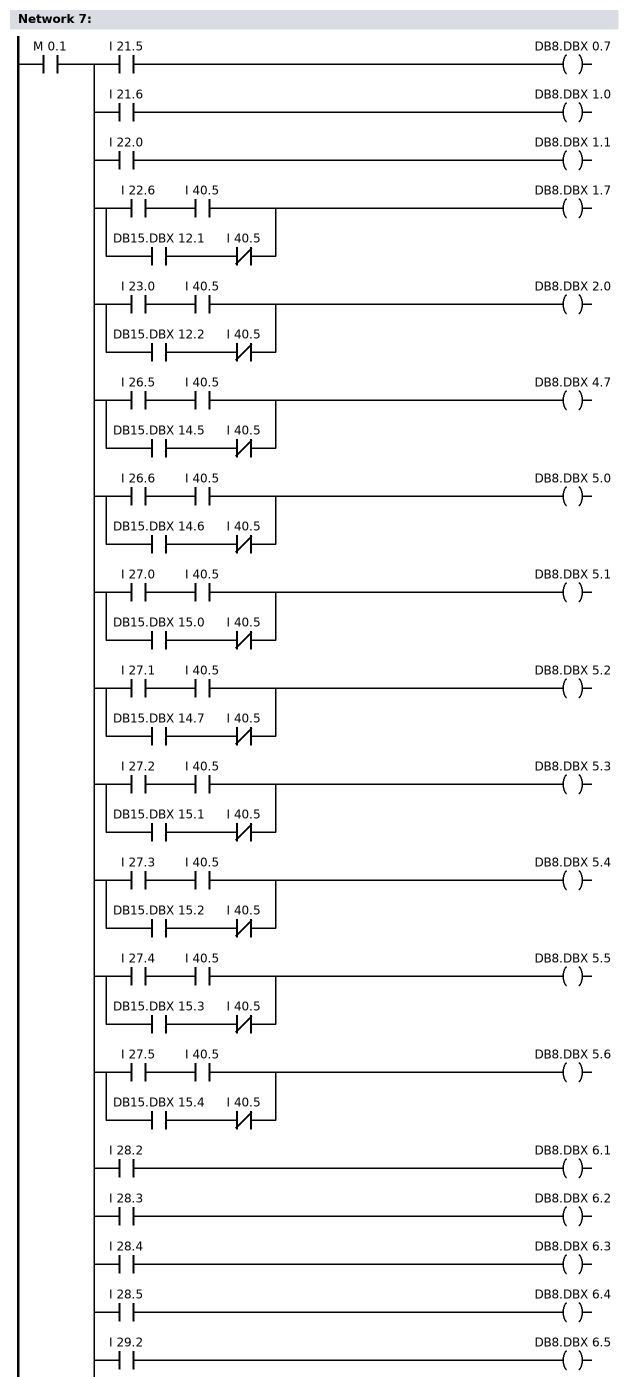
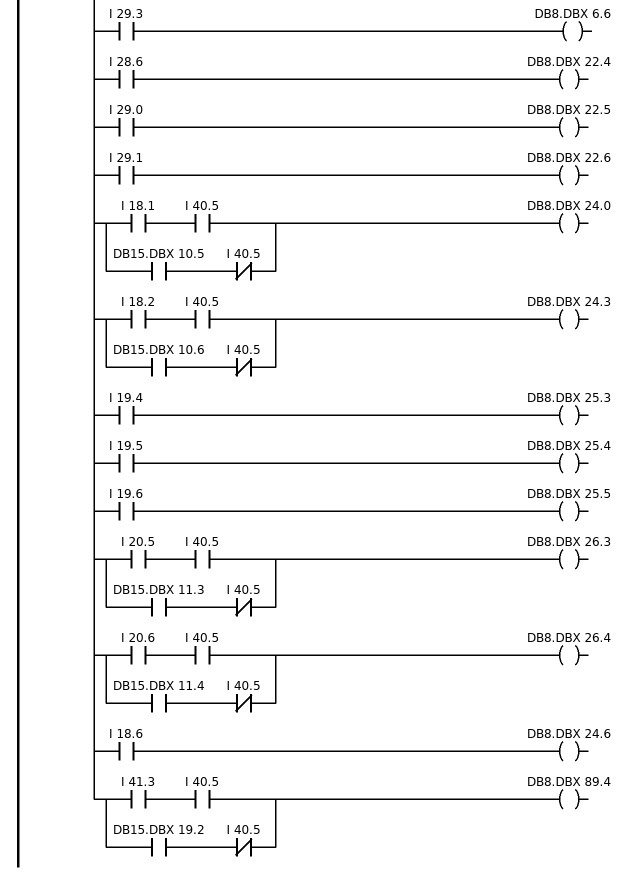
NETWORK
TITLE =
      A     M 0.1;
      =     L 0.0;
      A     L 0.0;
      A     I 21.5;
      =     DB8.DBX 0.7;
      A     L 0.0;
      A     I 21.6;
      =     DB8.DBX 1.0;
      A     L 0.0;
      A     I 22.0;
      =     DB8.DBX 1.1;
      A     L 0.0;
      A(;
      A     I 22.6;
      A     I 40.5;
      O;
      A     DB15.DBX 12.1;
      AN    I 40.5;
      );
      =     DB8.DBX 1.7;
      A     L 0.0;
      A(;
      A     I 23.0;
      A     I 40.5;
      O;
      A     DB15.DBX 12.2;
      AN    I 40.5;
      );
      =     DB8.DBX 2.0;
      A     L 0.0;
      A(;
      A     I 26.5;
      A     I 40.5;
      O;
      A     DB15.DBX 14.5;
      AN    I 40.5;
      );
      =     DB8.DBX 4.7;
      A     L 0.0;
      A(;
      A     I 26.6;
      A     I 40.5;
      O;
      A     DB15.DBX 14.6;
      AN    I 40.5;
      );
      =     DB8.DBX 5.0;
      A     L 0.0;
      A(;
      A     I 27.0;
      A     I 40.5;
      O;
      A     DB15.DBX 15.0;
      AN    I 40.5;
      );
      =     DB8.DBX 5.1;
      A     L 0.0;
      A(;
      A     I 27.1;
      A     I 40.5;
      O;
      A     DB15.DBX 14.7;
      AN    I 40.5;
      );
      =     DB8.DBX 5.2;
      A     L 0.0;
      A(;
      A     I 27.2;
      A     I 40.5;
      O;
      A     DB15.DBX 15.1;
      AN    I 40.5;
      );
      =     DB8.DBX 5.3;
      A     L 0.0;
      A(;
      A     I 27.3;
      A     I 40.5;
      O;
      A     DB15.DBX 15.2;
      AN    I 40.5;
      );
      =     DB8.DBX 5.4;
      A     L 0.0;
      A(;
      A     I 27.4;
      A     I 40.5;
      O;
      A     DB15.DBX 15.3;
      AN    I 40.5;
      );
      =     DB8.DBX 5.5;
      A     L 0.0;
      A(;
      A     I 27.5;
      A     I 40.5;
      O;
      A     DB15.DBX 15.4;
      AN    I 40.5;
      );
      =     DB8.DBX 5.6;
      A     L 0.0;
      A     I 28.2;
      =     DB8.DBX 6.1;
      A     L 0.0;
      A     I 28.3;
      =     DB8.DBX 6.2;
      A     L 0.0;
      A     I 28.4;
      =     DB8.DBX 6.3;
      A     L 0.0;
      A     I 28.5;
      =     DB8.DBX 6.4;
      A     L 0.0;
      A     I 29.2;
      =     DB8.DBX 6.5;
      A     L 0.0;
      A     I 29.3;
      =     DB8.DBX 6.6;
      A     L 0.0;
      A     I 28.6;
      =     DB8.DBX 22.4;
      A     L 0.0;
      A     I 29.0;
      =     DB8.DBX 22.5;
      A     L 0.0;
      A     I 29.1;
      =     DB8.DBX 22.6;
      A     L 0.0;
      A(;
      A     I 18.1;
      A     I 40.5;
      O;
      A     DB15.DBX 10.5;
      AN    I 40.5;
      );
      =     DB8.DBX 24.0;
      A     L 0.0;
      A(;
      A     I 18.2;
      A     I 40.5;
      O;
      A     DB15.DBX 10.6;
      AN    I 40.5;
      );
      =     DB8.DBX 24.3;
      A     L 0.0;
      A     I 19.4;
      =     DB8.DBX 25.3;
      A     L 0.0;
      A     I 19.5;
      =     DB8.DBX 25.4;
      A     L 0.0;
      A     I 19.6;
      =     DB8.DBX 25.5;
      A     L 0.0;
      A(;
      A     I 20.5;
      A     I 40.5;
      O;
      A     DB15.DBX 11.3;
      AN    I 40.5;
      );
      =     DB8.DBX 26.3;
      A     L 0.0;
      A(;
      A     I 20.6;
      A     I 40.5;
      O;
      A     DB15.DBX 11.4;
      AN    I 40.5;
      );
      =     DB8.DBX 26.4;
      A     L 0.0;
      A     I 18.6;
      =     DB8.DBX 24.6;
      A     L 0.0;
      A(;
      A     I 41.3;
      A     I 40.5;
      O;
      A     DB15.DBX 19.2;
      AN    I 40.5;
      );
      =     DB8.DBX 89.4;
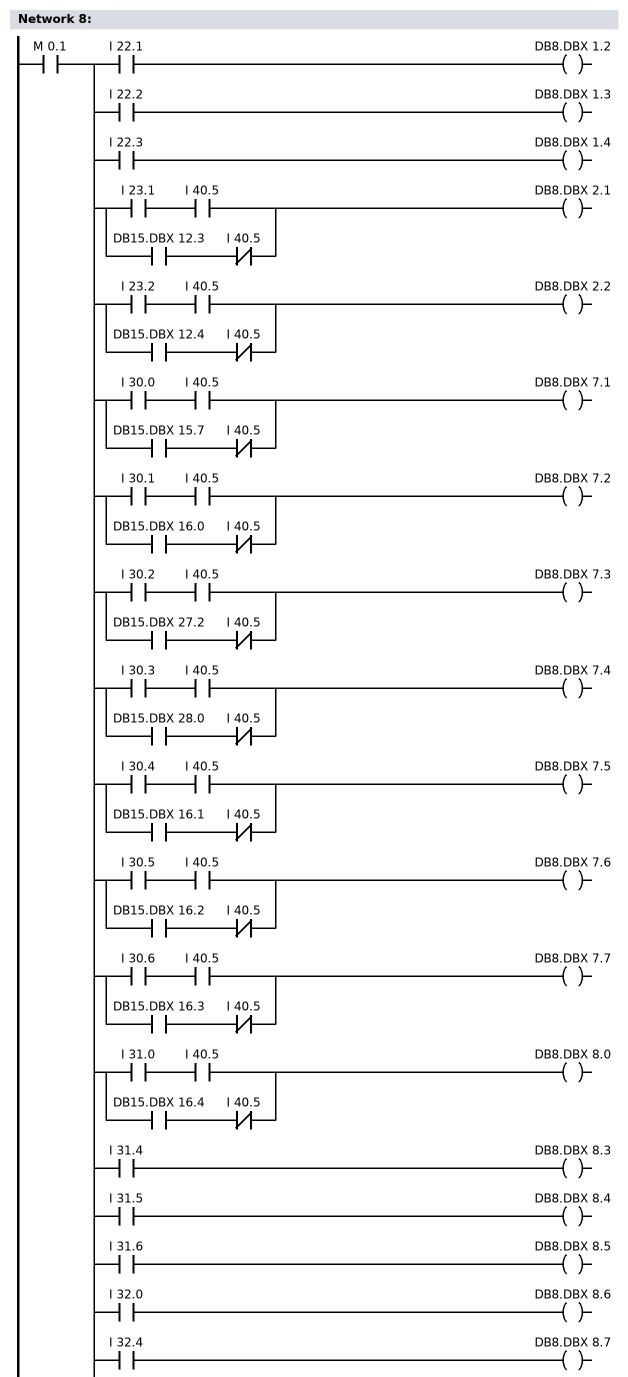
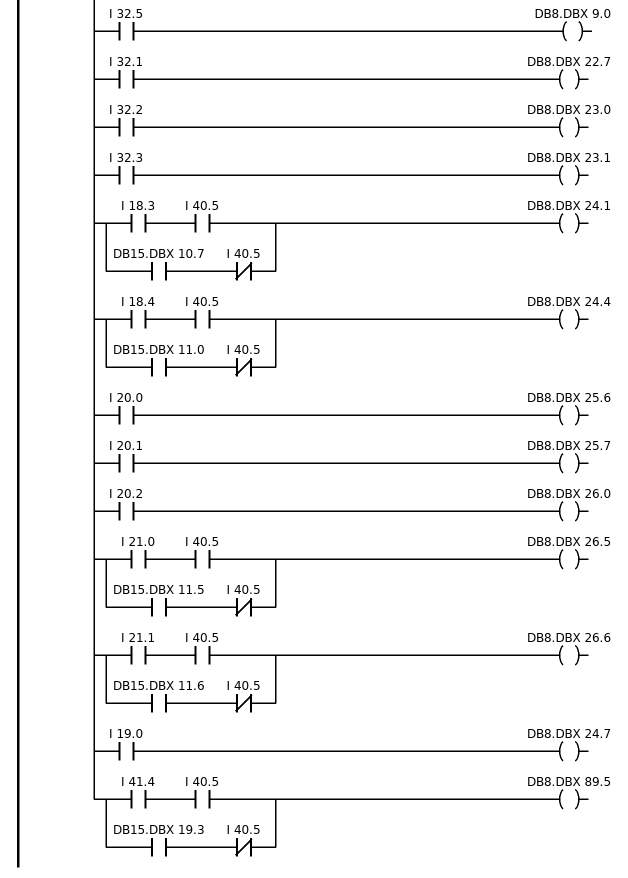
NETWORK
TITLE =
      A     M 0.1;
      =     L 0.0;
      A     L 0.0;
      A     I 22.1;
      =     DB8.DBX 1.2;
      A     L 0.0;
      A     I 22.2;
      =     DB8.DBX 1.3;
      A     L 0.0;
      A     I 22.3;
      =     DB8.DBX 1.4;
      A     L 0.0;
      A(;
      A     I 23.1;
      A     I 40.5;
      O;
      A     DB15.DBX 12.3;
      AN    I 40.5;
      );
      =     DB8.DBX 2.1;
      A     L 0.0;
      A(;
      A     I 23.2;
      A     I 40.5;
      O;
      A     DB15.DBX 12.4;
      AN    I 40.5;
      );
      =     DB8.DBX 2.2;
      A     L 0.0;
      A(;
      A     I 30.0;
      A     I 40.5;
      O;
      A     DB15.DBX 15.7;
      AN    I 40.5;
      );
      =     DB8.DBX 7.1;
      A     L 0.0;
      A(;
      A     I 30.1;
      A     I 40.5;
      O;
      A     DB15.DBX 16.0;
      AN    I 40.5;
      );
      =     DB8.DBX 7.2;
      A     L 0.0;
      A(;
      A     I 30.2;
      A     I 40.5;
      O;
      A     DB15.DBX 27.2;
      AN    I 40.5;
      );
      =     DB8.DBX 7.3;
      A     L 0.0;
      A(;
      A     I 30.3;
      A     I 40.5;
      O;
      A     DB15.DBX 28.0;
      AN    I 40.5;
      );
      =     DB8.DBX 7.4;
      A     L 0.0;
      A(;
      A     I 30.4;
      A     I 40.5;
      O;
      A     DB15.DBX 16.1;
      AN    I 40.5;
      );
      =     DB8.DBX 7.5;
      A     L 0.0;
      A(;
      A     I 30.5;
      A     I 40.5;
      O;
      A     DB15.DBX 16.2;
      AN    I 40.5;
      );
      =     DB8.DBX 7.6;
      A     L 0.0;
      A(;
      A     I 30.6;
      A     I 40.5;
      O;
      A     DB15.DBX 16.3;
      AN    I 40.5;
      );
      =     DB8.DBX 7.7;
      A     L 0.0;
      A(;
      A     I 31.0;
      A     I 40.5;
      O;
      A     DB15.DBX 16.4;
      AN    I 40.5;
      );
      =     DB8.DBX 8.0;
      A     L 0.0;
      A     I 31.4;
      =     DB8.DBX 8.3;
      A     L 0.0;
      A     I 31.5;
      =     DB8.DBX 8.4;
      A     L 0.0;
      A     I 31.6;
      =     DB8.DBX 8.5;
      A     L 0.0;
      A     I 32.0;
      =     DB8.DBX 8.6;
      A     L 0.0;
      A     I 32.4;
      =     DB8.DBX 8.7;
      A     L 0.0;
      A     I 32.5;
      =     DB8.DBX 9.0;
      A     L 0.0;
      A     I 32.1;
      =     DB8.DBX 22.7;
      A     L 0.0;
      A     I 32.2;
      =     DB8.DBX 23.0;
      A     L 0.0;
      A     I 32.3;
      =     DB8.DBX 23.1;
      A     L 0.0;
      A(;
      A     I 18.3;
      A     I 40.5;
      O;
      A     DB15.DBX 10.7;
      AN    I 40.5;
      );
      =     DB8.DBX 24.1;
      A     L 0.0;
      A(;
      A     I 18.4;
      A     I 40.5;
      O;
      A     DB15.DBX 11.0;
      AN    I 40.5;
      );
      =     DB8.DBX 24.4;
      A     L 0.0;
      A     I 20.0;
      =     DB8.DBX 25.6;
      A     L 0.0;
      A     I 20.1;
      =     DB8.DBX 25.7;
      A     L 0.0;
      A     I 20.2;
      =     DB8.DBX 26.0;
      A     L 0.0;
      A(;
      A     I 21.0;
      A     I 40.5;
      O;
      A     DB15.DBX 11.5;
      AN    I 40.5;
      );
      =     DB8.DBX 26.5;
      A     L 0.0;
      A(;
      A     I 21.1;
      A     I 40.5;
      O;
      A     DB15.DBX 11.6;
      AN    I 40.5;
      );
      =     DB8.DBX 26.6;
      A     L 0.0;
      A     I 19.0;
      =     DB8.DBX 24.7;
      A     L 0.0;
      A(;
      A     I 41.4;
      A     I 40.5;
      O;
      A     DB15.DBX 19.3;
      AN    I 40.5;
      );
      =     DB8.DBX 89.5;
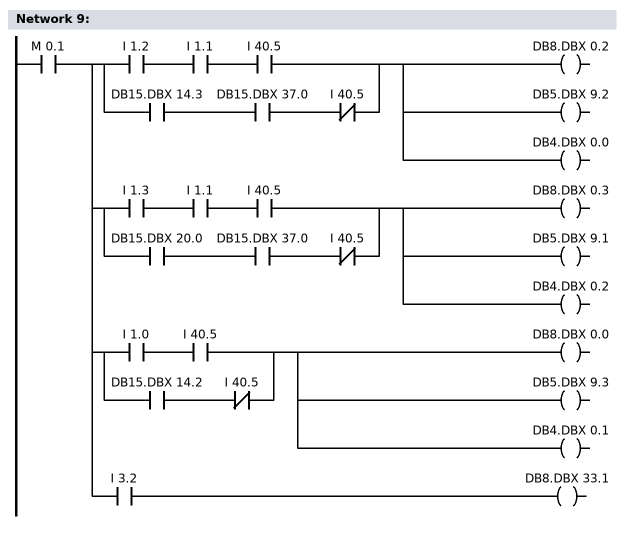
NETWORK
TITLE =
      A     M 0.1;
      =     L 0.0;
      A     L 0.0;
      A(;
      A     I 1.2;
      A     I 1.1;
      A     I 40.5;
      O;
      A     DB15.DBX 14.3;
      A     DB15.DBX 37.0;
      AN    I 40.5;
      );
      =     DB8.DBX 0.2;
      =     DB5.DBX 9.2;
      =     DB4.DBX 0.0;
      A     L 0.0;
      A(;
      A     I 1.3;
      A     I 1.1;
      A     I 40.5;
      O;
      A     DB15.DBX 20.0;
      A     DB15.DBX 37.0;
      AN    I 40.5;
      );
      =     DB8.DBX 0.3;
      =     DB5.DBX 9.1;
      =     DB4.DBX 0.2;
      A     L 0.0;
      A(;
      A     I 1.0;
      A     I 40.5;
      O;
      A     DB15.DBX 14.2;
      AN    I 40.5;
      );
      =     DB8.DBX 0.0;
      =     DB5.DBX 9.3;
      =     DB4.DBX 0.1;
      A     L 0.0;
      A     I 3.2;
      =     DB8.DBX 33.1;
END_FUNCTION

FUNCTION FC 6 : VOID
AUTHOR : Arun_Ram
VERSION : 0.1
BEGIN
// (block stored without names or comments; labels and parameter names are numbered)
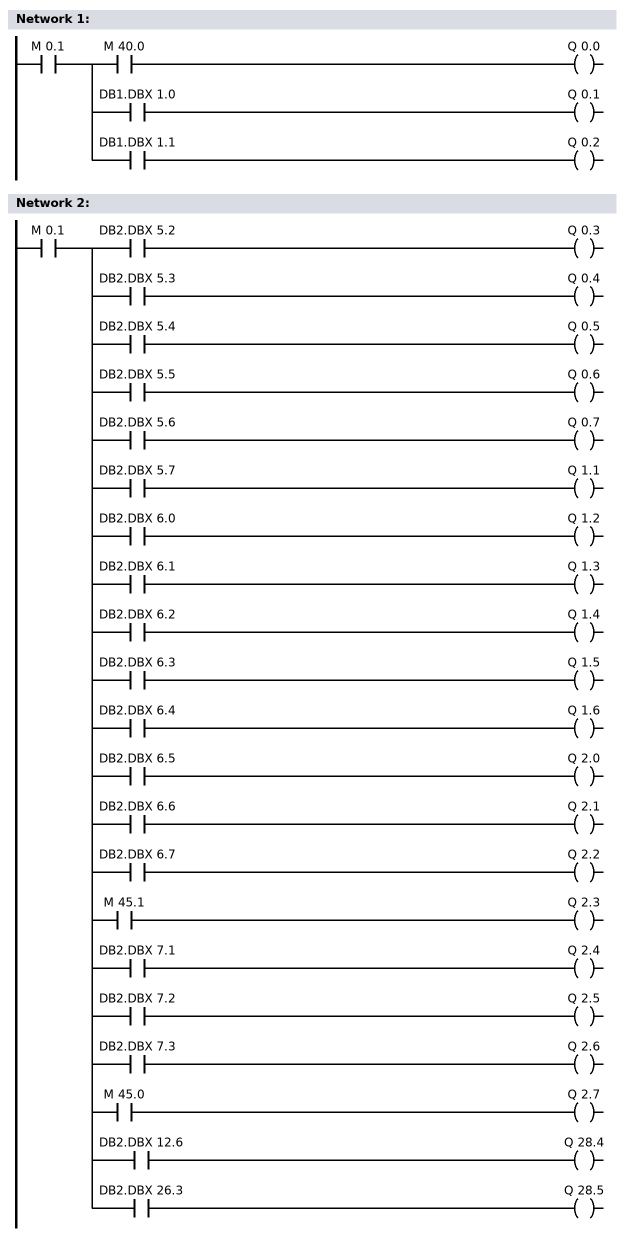
NETWORK
TITLE =
      A     M 0.1;
      =     L 0.0;
      A     L 0.0;
      A     M 40.0;
      =     Q 0.0;
      A     L 0.0;
      A     DB1.DBX 1.0;
      =     Q 0.1;
      A     L 0.0;
      A     DB1.DBX 1.1;
      =     Q 0.2;
NETWORK
TITLE =
      A     M 0.1;
      =     L 0.0;
      A     L 0.0;
      A     DB2.DBX 5.2;
      =     Q 0.3;
      A     L 0.0;
      A     DB2.DBX 5.3;
      =     Q 0.4;
      A     L 0.0;
      A     DB2.DBX 5.4;
      =     Q 0.5;
      A     L 0.0;
      A     DB2.DBX 5.5;
      =     Q 0.6;
      A     L 0.0;
      A     DB2.DBX 5.6;
      =     Q 0.7;
      A     L 0.0;
      A     DB2.DBX 5.7;
      =     Q 1.1;
      A     L 0.0;
      A     DB2.DBX 6.0;
      =     Q 1.2;
      A     L 0.0;
      A     DB2.DBX 6.1;
      =     Q 1.3;
      A     L 0.0;
      A     DB2.DBX 6.2;
      =     Q 1.4;
      A     L 0.0;
      A     DB2.DBX 6.3;
      =     Q 1.5;
      A     L 0.0;
      A     DB2.DBX 6.4;
      =     Q 1.6;
      A     L 0.0;
      A     DB2.DBX 6.5;
      =     Q 2.0;
      A     L 0.0;
      A     DB2.DBX 6.6;
      =     Q 2.1;
      A     L 0.0;
      A     DB2.DBX 6.7;
      =     Q 2.2;
      A     L 0.0;
      A     M 45.1;
      =     Q 2.3;
      A     L 0.0;
      A     DB2.DBX 7.1;
      =     Q 2.4;
      A     L 0.0;
      A     DB2.DBX 7.2;
      =     Q 2.5;
      A     L 0.0;
      A     DB2.DBX 7.3;
      =     Q 2.6;
      A     L 0.0;
      A     M 45.0;
      =     Q 2.7;
      A     L 0.0;
      A     DB2.DBX 12.6;
      =     Q 28.4;
      A     L 0.0;
      A     DB2.DBX 26.3;
      =     Q 28.5;
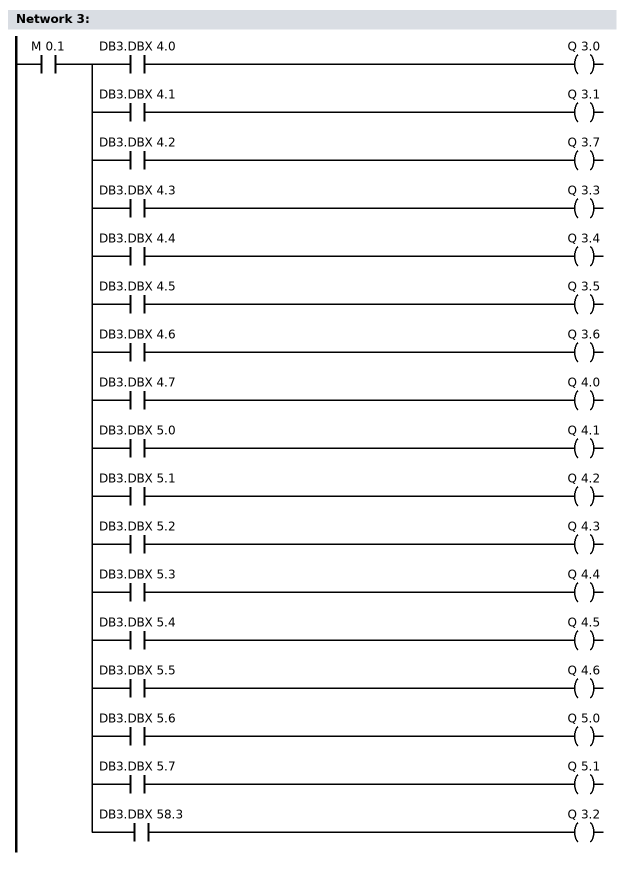
NETWORK
TITLE =
      A     M 0.1;
      =     L 0.0;
      A     L 0.0;
      A     DB3.DBX 4.0;
      =     Q 3.0;
      A     L 0.0;
      A     DB3.DBX 4.1;
      =     Q 3.1;
      A     L 0.0;
      A     DB3.DBX 4.2;
      =     Q 3.7;
      A     L 0.0;
      A     DB3.DBX 4.3;
      =     Q 3.3;
      A     L 0.0;
      A     DB3.DBX 4.4;
      =     Q 3.4;
      A     L 0.0;
      A     DB3.DBX 4.5;
      =     Q 3.5;
      A     L 0.0;
      A     DB3.DBX 4.6;
      =     Q 3.6;
      A     L 0.0;
      A     DB3.DBX 4.7;
      =     Q 4.0;
      A     L 0.0;
      A     DB3.DBX 5.0;
      =     Q 4.1;
      A     L 0.0;
      A     DB3.DBX 5.1;
      =     Q 4.2;
      A     L 0.0;
      A     DB3.DBX 5.2;
      =     Q 4.3;
      A     L 0.0;
      A     DB3.DBX 5.3;
      =     Q 4.4;
      A     L 0.0;
      A     DB3.DBX 5.4;
      =     Q 4.5;
      A     L 0.0;
      A     DB3.DBX 5.5;
      =     Q 4.6;
      A     L 0.0;
      A     DB3.DBX 5.6;
      =     Q 5.0;
      A     L 0.0;
      A     DB3.DBX 5.7;
      =     Q 5.1;
      A     L 0.0;
      A     DB3.DBX 58.3;
      =     Q 3.2;
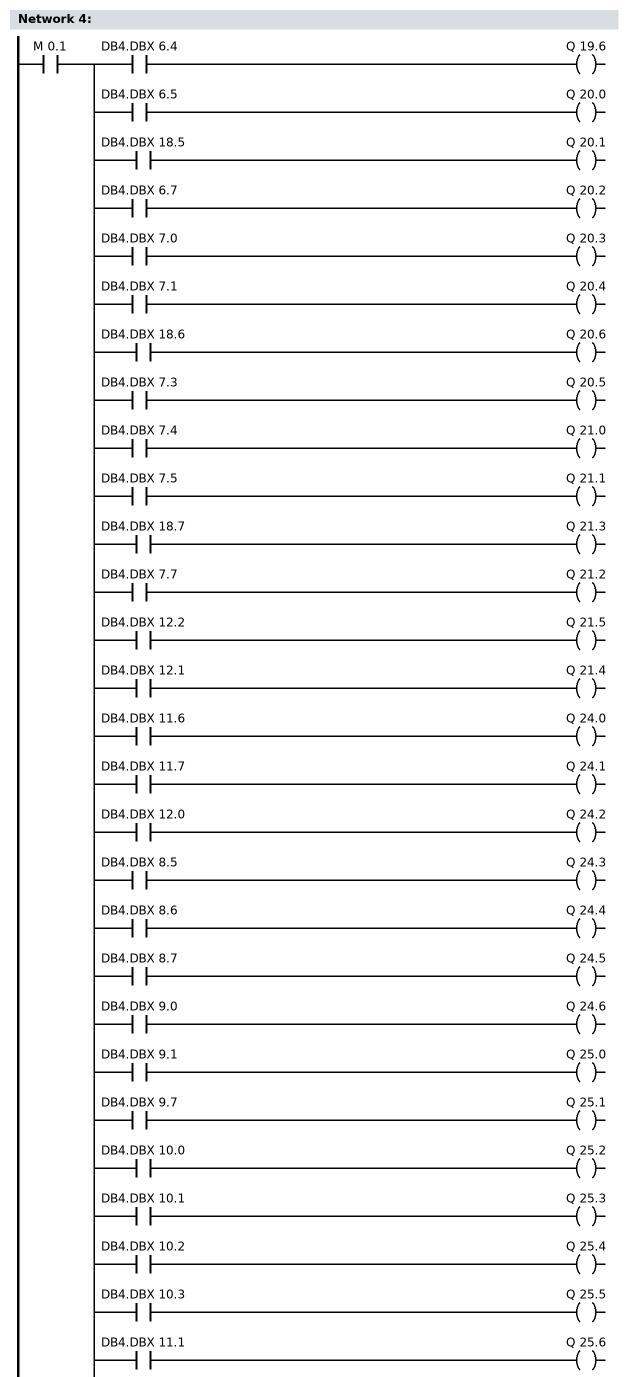
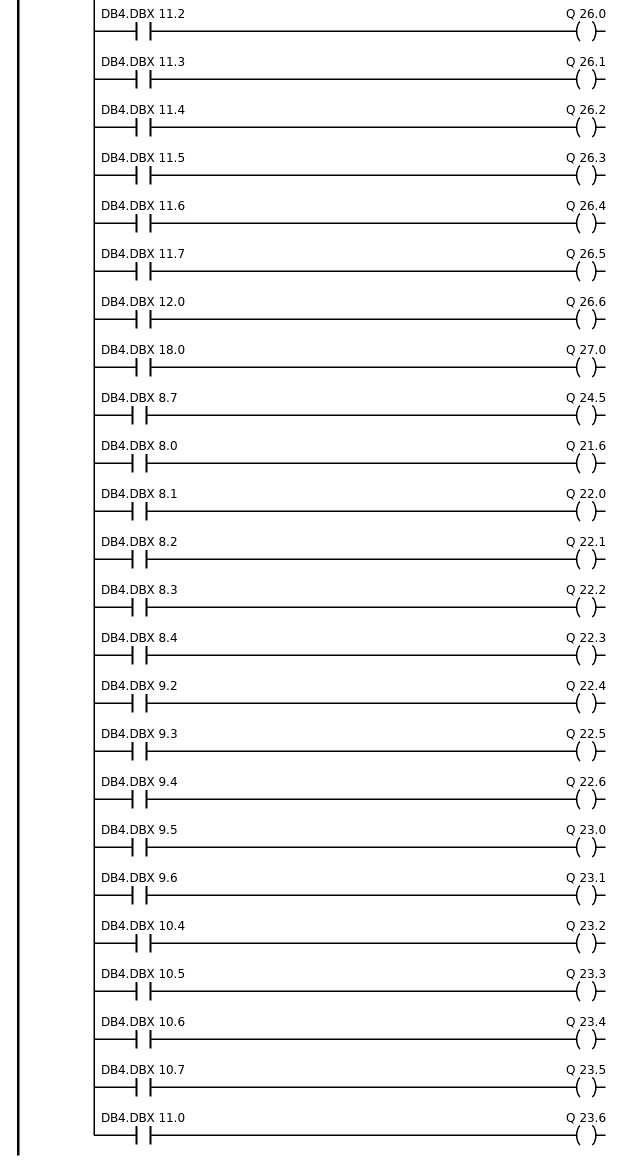
NETWORK
TITLE =
      A     M 0.1;
      =     L 0.0;
      A     L 0.0;
      A     DB4.DBX 6.4;
      =     Q 19.6;
      A     L 0.0;
      A     DB4.DBX 6.5;
      =     Q 20.0;
      A     L 0.0;
      A     DB4.DBX 18.5;
      =     Q 20.1;
      A     L 0.0;
      A     DB4.DBX 6.7;
      =     Q 20.2;
      A     L 0.0;
      A     DB4.DBX 7.0;
      =     Q 20.3;
      A     L 0.0;
      A     DB4.DBX 7.1;
      =     Q 20.4;
      A     L 0.0;
      A     DB4.DBX 18.6;
      =     Q 20.6;
      A     L 0.0;
      A     DB4.DBX 7.3;
      =     Q 20.5;
      A     L 0.0;
      A     DB4.DBX 7.4;
      =     Q 21.0;
      A     L 0.0;
      A     DB4.DBX 7.5;
      =     Q 21.1;
      A     L 0.0;
      A     DB4.DBX 18.7;
      =     Q 21.3;
      A     L 0.0;
      A     DB4.DBX 7.7;
      =     Q 21.2;
      A     L 0.0;
      A     DB4.DBX 12.2;
      =     Q 21.5;
      A     L 0.0;
      A     DB4.DBX 12.1;
      =     Q 21.4;
      A     L 0.0;
      A     DB4.DBX 11.6;
      =     Q 24.0;
      A     L 0.0;
      A     DB4.DBX 11.7;
      =     Q 24.1;
      A     L 0.0;
      A     DB4.DBX 12.0;
      =     Q 24.2;
      A     L 0.0;
      A     DB4.DBX 8.5;
      =     Q 24.3;
      A     L 0.0;
      A     DB4.DBX 8.6;
      =     Q 24.4;
      A     L 0.0;
      A     DB4.DBX 8.7;
      =     Q 24.5;
      A     L 0.0;
      A     DB4.DBX 9.0;
      =     Q 24.6;
      A     L 0.0;
      A     DB4.DBX 9.1;
      =     Q 25.0;
      A     L 0.0;
      A     DB4.DBX 9.7;
      =     Q 25.1;
      A     L 0.0;
      A     DB4.DBX 10.0;
      =     Q 25.2;
      A     L 0.0;
      A     DB4.DBX 10.1;
      =     Q 25.3;
      A     L 0.0;
      A     DB4.DBX 10.2;
      =     Q 25.4;
      A     L 0.0;
      A     DB4.DBX 10.3;
      =     Q 25.5;
      A     L 0.0;
      A     DB4.DBX 11.1;
      =     Q 25.6;
      A     L 0.0;
      A     DB4.DBX 11.2;
      =     Q 26.0;
      A     L 0.0;
      A     DB4.DBX 11.3;
      =     Q 26.1;
      A     L 0.0;
      A     DB4.DBX 11.4;
      =     Q 26.2;
      A     L 0.0;
      A     DB4.DBX 11.5;
      =     Q 26.3;
      A     L 0.0;
      A     DB4.DBX 11.6;
      =     Q 26.4;
      A     L 0.0;
      A     DB4.DBX 11.7;
      =     Q 26.5;
      A     L 0.0;
      A     DB4.DBX 12.0;
      =     Q 26.6;
      A     L 0.0;
      A     DB4.DBX 18.0;
      =     Q 27.0;
      A     L 0.0;
      A     DB4.DBX 8.7;
      =     Q 24.5;
      A     L 0.0;
      A     DB4.DBX 8.0;
      =     Q 21.6;
      A     L 0.0;
      A     DB4.DBX 8.1;
      =     Q 22.0;
      A     L 0.0;
      A     DB4.DBX 8.2;
      =     Q 22.1;
      A     L 0.0;
      A     DB4.DBX 8.3;
      =     Q 22.2;
      A     L 0.0;
      A     DB4.DBX 8.4;
      =     Q 22.3;
      A     L 0.0;
      A     DB4.DBX 9.2;
      =     Q 22.4;
      A     L 0.0;
      A     DB4.DBX 9.3;
      =     Q 22.5;
      A     L 0.0;
      A     DB4.DBX 9.4;
      =     Q 22.6;
      A     L 0.0;
      A     DB4.DBX 9.5;
      =     Q 23.0;
      A     L 0.0;
      A     DB4.DBX 9.6;
      =     Q 23.1;
      A     L 0.0;
      A     DB4.DBX 10.4;
      =     Q 23.2;
      A     L 0.0;
      A     DB4.DBX 10.5;
      =     Q 23.3;
      A     L 0.0;
      A     DB4.DBX 10.6;
      =     Q 23.4;
      A     L 0.0;
      A     DB4.DBX 10.7;
      =     Q 23.5;
      A     L 0.0;
      A     DB4.DBX 11.0;
      =     Q 23.6;
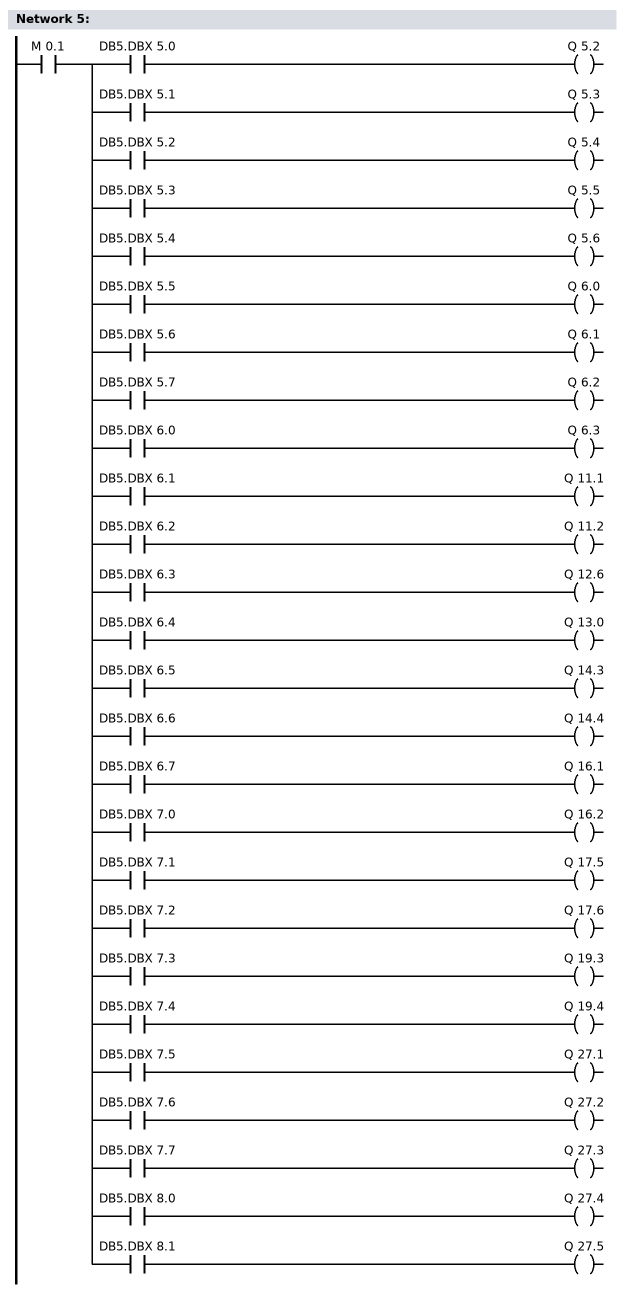
NETWORK
TITLE =
      A     M 0.1;
      =     L 0.0;
      A     L 0.0;
      A     DB5.DBX 5.0;
      =     Q 5.2;
      A     L 0.0;
      A     DB5.DBX 5.1;
      =     Q 5.3;
      A     L 0.0;
      A     DB5.DBX 5.2;
      =     Q 5.4;
      A     L 0.0;
      A     DB5.DBX 5.3;
      =     Q 5.5;
      A     L 0.0;
      A     DB5.DBX 5.4;
      =     Q 5.6;
      A     L 0.0;
      A     DB5.DBX 5.5;
      =     Q 6.0;
      A     L 0.0;
      A     DB5.DBX 5.6;
      =     Q 6.1;
      A     L 0.0;
      A     DB5.DBX 5.7;
      =     Q 6.2;
      A     L 0.0;
      A     DB5.DBX 6.0;
      =     Q 6.3;
      A     L 0.0;
      A     DB5.DBX 6.1;
      =     Q 11.1;
      A     L 0.0;
      A     DB5.DBX 6.2;
      =     Q 11.2;
      A     L 0.0;
      A     DB5.DBX 6.3;
      =     Q 12.6;
      A     L 0.0;
      A     DB5.DBX 6.4;
      =     Q 13.0;
      A     L 0.0;
      A     DB5.DBX 6.5;
      =     Q 14.3;
      A     L 0.0;
      A     DB5.DBX 6.6;
      =     Q 14.4;
      A     L 0.0;
      A     DB5.DBX 6.7;
      =     Q 16.1;
      A     L 0.0;
      A     DB5.DBX 7.0;
      =     Q 16.2;
      A     L 0.0;
      A     DB5.DBX 7.1;
      =     Q 17.5;
      A     L 0.0;
      A     DB5.DBX 7.2;
      =     Q 17.6;
      A     L 0.0;
      A     DB5.DBX 7.3;
      =     Q 19.3;
      A     L 0.0;
      A     DB5.DBX 7.4;
      =     Q 19.4;
      A     L 0.0;
      A     DB5.DBX 7.5;
      =     Q 27.1;
      A     L 0.0;
      A     DB5.DBX 7.6;
      =     Q 27.2;
      A     L 0.0;
      A     DB5.DBX 7.7;
      =     Q 27.3;
      A     L 0.0;
      A     DB5.DBX 8.0;
      =     Q 27.4;
      A     L 0.0;
      A     DB5.DBX 8.1;
      =     Q 27.5;
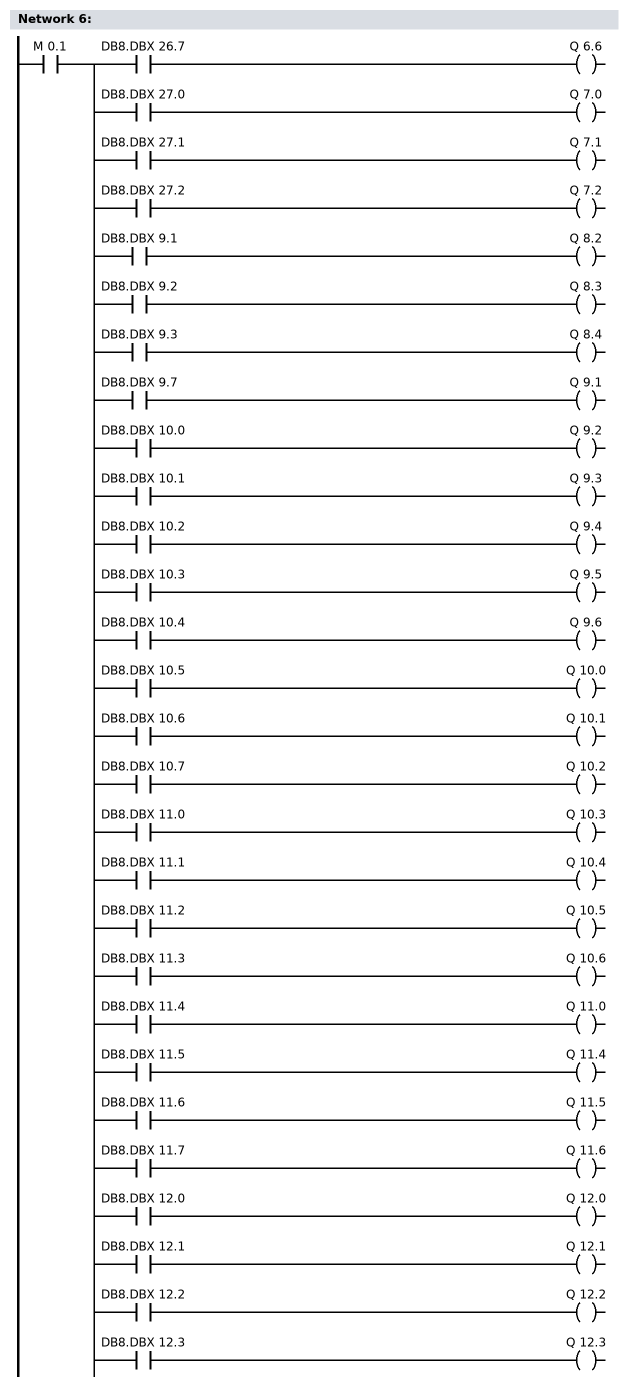
